E_MachineState.IMMEDIATE_STOPPED:	
	(* Move to System Initialising once there is no Immediate Fault *)
	IF GVL_MASTER.stMasterControl.bNoMachineImmediateFault  THEN	
		GVL_MASTER.stMachineStatus.eMachineState := E_MachineState.SYSTEM_INITIALISING;
	(* Move to Immediate Fault once there is an Immediate Fault *)
	ELSIF NOT GVL_MASTER.stMasterControl.bNoMachineImmediateFault THEN
		GVL_MASTER.stMachineStatus.eMachineState := E_MachineState.IMMEDIATE_FAULT;	
	END_IF
	
E_MachineState.SYSTEM_INITIALISING:		
	IF  GVL_MASTER.stMasterControl.bNoMachineImmediateFault	 AND GVL_MASTER.stMasterControl.bSystemInitialisingTimerComplete  THEN		
		GVL_MASTER.stMachineStatus.eMachineState := E_MachineState.SYSTEM_READY_TO_START;
	
	//Move to Cycle Stopped once there is a Cycle Stop Request AND All Stations are Cycle Stopped AND there is No Immediate Fault*)
	ELSIF GVL_HMI_GLOBAL.bStopButton
		OR (GVL_MASTER.stMasterControl.bNoMachineImmediateFault 
		AND (GVL_MASTER.stMasterControl.bSystemInitialisingTimeoutComplete OR GVL_MASTER.stMasterControl.bCycleStopRequest) AND GVL_MASTER.stMasterControl.bAllStationsCycledStopped)
	THEN		
		GVL_MASTER.stMachineStatus.eMachineState := E_MachineState.CYCLE_STOPPED;			
	ELSIF GVL_MASTER.stMasterControl.bNoMachineImmediateFault AND NOT GVL_MASTER.stMasterControl.bNoCycleStopFault THEN		
		GVL_MASTER.stMachineStatus.eMachineState := E_MachineState.CYCLE_STOP_FAULT;	
	ELSIF NOT GVL_MASTER.stMasterControl.bNoStationImmediateFault THEN
         GVL_MASTER.stMachineStatus.eMachineState := E_MachineState.IMMEDIATE_FAULT;
      	
	END_IF
	
E_MachineState.SYSTEM_READY_TO_START:
	bMemoSystemReadyToStart := TRUE;
	
	//Move to System Auto if the Start Button has been pressed
	IF GVL_MASTER.stMasterControl.bManualModeRequest THEN
		GVL_MASTER.stMachineStatus.eMachineState := E_MachineState.MANUAL_MODE;
	
	ELSIF GVL_HMI_GLOBAL.bStopButton THEN
        GVL_MASTER.stMachineStatus.eMachineState := E_MachineState.STOPPING; 
	ELSIF GVL_HMI_GLOBAL.bStartButton AND NOT PRG_Mastercycle.biClamp AND NOT PRG_Mastercycle.biPartPresent  THEN		//**LAA 18092025	
		GVL_MASTER.stMachineStatus.eMachineState := E_MachineState.SYSTEM_AUTO_CYCLE;
		
	//Move to Cycle Stopped once there is a Cycle Stop Request AND All Stations are Cycle Stopped AND there is No Immediate Fault
	ELSIF (GVL_MASTER.stMasterControl.bCycleStopRequest OR NOT	GVL_MASTER.stMasterControl.bNoCycleStopFault) 
	AND GVL_MASTER.stMasterControl.bNoMachineImmediateFault
	THEN				
		GVL_MASTER.stMachineStatus.eMachineState := E_MachineState.CYCLE_STOPPED;	
	ELSIF NOT GVL_MASTER.stMasterControl.bNoCycleStopFault THEN
		GVL_MASTER.stMachineStatus.eMachineState := E_MachineState.CYCLE_STOP_FAULT;
	ELSIF NOT GVL_MASTER.stMasterControl.bNoMachineImmediateFault OR NOT GVL_MASTER.stMasterControl.bNoStationImmediateFault THEN
       GVL_MASTER.stMachineStatus.eMachineState := E_MachineState.IMMEDIATE_FAULT ;	
	   
	END_IF
	

	
	
	
E_MachineState.SYSTEM_AUTO_CYCLE:	
	//Move to System Dwell once there is a Dwell Request
	IF GVL_MASTER.stMasterControl.bDwellRequest THEN
		GVL_MASTER.stMachineStatus.eMachineState := E_MachineState.SYSTEM_DWELL;
	
	//Move to Cycle Stopped once there is a Cycle Stop Request AND All Stations are Cycle Stopped AND there is No Immediate Fault OR when cycle done
	ELSIF NOT GVL_MASTER.stMasterControl.bNoCycleStopFault THEN //Fast cycle stop	
		GVL_MASTER.stMachineStatus.eMachineState := E_MachineState.CYCLE_STOP_FAULT;
	(*ELSIF GVL_Master.bMachineCycleDone   THEN 
	stMachineStatus.eMachineState := E_MachineState.CYCLE_STOPPED; //Instant cycle stop???		*)
	ELSIF GVL_HMI_GLOBAL.bStopButton OR GVL_MASTER.stMasterControl.bCycleStopRequest OR GVL_HMI_GLOBAL.nRegionMain <> 1 THEN
		GVL_MASTER.stMachineStatus.eMachineState := E_MachineState.STOPPING; //Stopping sequence 
	ELSIF NOT GVL_MASTER.stMasterControl.bNoStationImmediateFault OR NOT GVL_MASTER.stMasterControl.bNoMachineImmediateFault THEN
		GVL_MASTER.stMachineStatus.eMachineState := E_MachineState.IMMEDIATE_FAULT;
	END_IF	

E_MachineState.SYSTEM_DWELL:		
	(* Move to System Auto Cycle once the Start Button is Pressed AND there is No Dwell Request *)
	IF NOT GVL_MASTER.stMasterControl.bDwellRequest THEN
		GVL_MASTER.stMachineStatus.eMachineState := E_MachineState.SYSTEM_AUTO_CYCLE;	
	(* Move to Cycle Stopped once there is a Cycle Stop Request AND All Stations are Cycle Stopped AND there is No Immediate Fault*)
	ELSIF (GVL_MASTER.stMasterControl.bCycleStopRequest OR	NOT	GVL_MASTER.stMasterControl.bNoCycleStopFault) 
		AND GVL_MASTER.stMasterControl.bAllStationsCycledStopped AND GVL_MASTER.stMasterControl.bNoMachineImmediateFault
	THEN				
		GVL_MASTER.stMachineStatus.eMachineState := E_MachineState.CYCLE_STOPPED;	
	END_IF

E_MachineState.STOPPING: 
	IF  GVL_MASTER.stMasterControl.bAllStationsCycledStopped THEN
		GVL_MASTER.stMachineStatus.eMachineState := E_MachineState.CYCLE_STOPPED;
	ELSIF NOT GVL_MASTER.stMasterControl.bNoCycleStopFault THEN
		GVL_MASTER.stMachineStatus.eMachineState := E_MachineState.CYCLE_STOP_FAULT;
	ELSIF NOT GVL_MASTER.stMasterControl.bNoMachineImmediateFault OR NOT GVL_MASTER.stMasterControl.bNoStationImmediateFault THEN
        GVL_MASTER.stMachineStatus.eMachineState := E_MachineState.IMMEDIATE_FAULT ;
	END_IF
	
E_MachineState.CYCLE_STOPPED:
	IF GVL_MASTER.stMasterControl.bManualModeRequest THEN
		GVL_MASTER.stMachineStatus.eMachineState := E_MachineState.MANUAL_MODE;			
	(* Move to System Initialising once there is no Cycle Stop Fault AND the Reset Button is Pressed *)
	ELSIF (GVL_MASTER.stMasterControl.bNoCycleStopFault AND GVL_HMI_GLOBAL.bResetButton )THEN
		GVL_MASTER.stMachineStatus.eMachineState := E_MachineState.SYSTEM_INITIALISING;		
	ELSIF NOT GVL_MASTER.stMasterControl.bNoStationImmediateFault THEN
       	GVL_MASTER.stMachineStatus.eMachineState := E_MachineState.IMMEDIATE_FAULT;
	END_IF	

E_MachineState.CYCLE_STOP_FAULT:	
	(* Move to Cycle Stopped once there no Cycle Stop Fault AND there is No Immediate Fault*)
	IF GVL_MASTER.stMasterControl.bNoCycleStopFault THEN
		GVL_MASTER.stMachineStatus.eMachineState := E_MachineState.CYCLE_STOPPED;
	END_IF	
ELSE 	
	GVL_MASTER.stMachineStatus.eMachineState := E_MachineState.SYSTEM_POWER_UP;	
	
E_MachineState.MANUAL_MODE:

	IF NOT GVL_MASTER.stMasterControl.bManualModeRequest THEN
		GVL_MASTER.stMachineStatus.eMachineState := E_MachineState.CYCLE_STOPPED;
	END_IF
	
E_MachineState.IMMEDIATE_FAULT:		
	(* Move to Immediate Stopped once there is an Immediate Fault *)
	IF GVL_MASTER.stMasterControl.bNoMachineImmediateFault AND  GVL_MASTER.stMasterControl.bNoStationImmediateFault THEN
		GVL_MASTER.stMachineStatus.eMachineState := E_MachineState.IMMEDIATE_STOPPED;		

	END_IF
END_CASE
//////////////////////////////////////////////////////////////////////////////////////////////////////////////
								//CYCLE STOP REQUEST//
//////////////////////////////////////////////////////////////////////////////////////////////////////////////
IF GVL_MASTER.stAlarms[0].bCycleStopRequest OR GVL_MASTER.stAlarms[1].bCycleStopRequest OR GVL_MASTER.stAlarms[2].bCycleStopRequest THEN
				GVL_MASTER.stMasterControl.bCycleStopRequest	:=	TRUE;
ELSE			GVL_MASTER.stMasterControl.bCycleStopRequest	:=	FALSE;
END_IF




(************************************* write all system states to variables ***********************)

GVL_MASTER.stMachineStatus.bSystemPowerUp :=(GVL_MASTER.stMachineStatus.eMachineState = E_MachineState.SYSTEM_POWER_UP);
GVL_MASTER.stMachineStatus.bImmediateStopped :=(GVL_MASTER.stMachineStatus.eMachineState = E_MachineState.IMMEDIATE_STOPPED);
GVL_MASTER.stMachineStatus.bSystemInitialising :=(GVL_MASTER.stMachineStatus.eMachineState = E_MachineState.SYSTEM_INITIALISING);
GVL_MASTER.stMachineStatus.bSystemReadyToStart := (GVL_MASTER.stMachineStatus.eMachineState = E_MachineState.SYSTEM_READY_TO_START);
GVL_MASTER.stMachineStatus.bSystemAutoCycle := (GVL_MASTER.stMachineStatus.eMachineState = E_MachineState.SYSTEM_AUTO_CYCLE);
GVL_MASTER.stMachineStatus.bSystemDwell := (GVL_MASTER.stMachineStatus.eMachineState = E_MachineState.SYSTEM_DWELL);
GVL_MASTER.stMachineStatus.bSystemStopping := (GVL_MASTER.stMachineStatus.eMachineState = E_MachineState.STOPPING);
GVL_MASTER.stMachineStatus.bCycleStopped := (GVL_MASTER.stMachineStatus.eMachineState = E_MachineState.CYCLE_STOPPED);
GVL_MASTER.stMachineStatus.bManualMode := (GVL_MASTER.stMachineStatus.eMachineState = E_MachineState.MANUAL_MODE);
GVL_MASTER.stMachineStatus.bImmediateFault := (GVL_MASTER.stMachineStatus.eMachineState = E_MachineState.IMMEDIATE_FAULT);
GVL_MASTER.stMachineStatus.bCycleStopFault := (GVL_MASTER.stMachineStatus.eMachineState = E_MachineState.CYCLE_STOP_FAULT);

ACTION ACT_MachineStatusBaner:
//Machine status banner action
//SYSTEM POWER UP
IF GVL_MASTER.stMachineStatus.bSystemPowerUp THEN	
	GVL_MASTER.stMachineStatus.sMachineStatusText := 'SYSTEM POWER UP';		// fill colour WHITE, text colour BLACK
	GVL_MASTER.stMachineStatus.nMachineStatusColour := nWHITE;
	GVL_MASTER.stMachineStatus.nMachineStatusTxtCol := nBLACK;
	GVL_MASTER.stMachineStatus.sBannerBckColor := sWHITE;
	GVL_MASTER.stMachineStatus.sBannerTextColor := sBLACK;
END_IF

(* IMMEDIATE STOPPED *)
IF GVL_MASTER.stMachineStatus.bImmediateStopped THEN	
	GVL_MASTER.stMachineStatus.sMachineStatusText := 'IMMEDIATE STOPPED';		// fill colour BLACK, text colour WHITE
	GVL_MASTER.stMachineStatus.nMachineStatusColour := nBLACK;
	GVL_MASTER.stMachineStatus.nMachineStatusTxtCol := nWHITE;
	GVL_MASTER.stMachineStatus.sBannerBckColor := sBLACK;
	GVL_MASTER.stMachineStatus.sBannerTextColor := sWHITE;	
END_IF

(* SYSTEM INITIALISING *)
IF GVL_MASTER.stMachineStatus.bSystemInitialising THEN	
	GVL_MASTER.stMachineStatus.sMachineStatusText := 'SYSTEM INITIALIZING';		// fill colour YELLOW, text colour BLACK
	GVL_MASTER.stMachineStatus.nMachineStatusColour := nYELLOW;
	GVL_MASTER.stMachineStatus.nMachineStatusTxtCol := nBLACK;
	GVL_MASTER.stMachineStatus.sBannerBckColor := sYELLOW;
	GVL_MASTER.stMachineStatus.sBannerTextColor := sBLACK;
END_IF
(*
(* SYSTEM IN STANDBY *)
IF stMachineStatus.bSystemStandby THEN
	stMachineStatus.sMachineStatusText := 'SYSTEM IN STANDBY';
	stMachineStatus.nMachineStatusColour := nORANGE;
	stMachineStatus.nMachineStatusTxtCol := nWHITE;
END_IF
*)
(* SYSTEM READY TO START FLASH ON *)
IF GVL_MASTER.stMachineStatus.bSystemReadyToStart AND GVL_MASTER.bFlash1Hz THEN
	GVL_MASTER.stMachineStatus.sMachineStatusText := 'SYSTEM READY TO START';		// fill colour GREEN, text colour WHITE
	GVL_MASTER.stMachineStatus.nMachineStatusColour := nGREEN;
	GVL_MASTER.stMachineStatus.nMachineStatusTxtCol := nWHITE;
	GVL_MASTER.stMachineStatus.sBannerBckColor := sGREEN;
	GVL_MASTER.stMachineStatus.sBannerTextColor := sWHITE;
END_IF

(* SYSTEM READY TO START FLASH OFF *)
IF GVL_MASTER.stMachineStatus.bSystemReadyToStart AND NOT GVL_MASTER.bFlash1Hz THEN	
	GVL_MASTER.stMachineStatus.sMachineStatusText := 'SYSTEM READY TO START';		// fill colour WHITE, text colour GREEN
	GVL_MASTER.stMachineStatus.nMachineStatusColour := nWHITE;
	GVL_MASTER.stMachineStatus.nMachineStatusTxtCol := nGREEN;
	GVL_MASTER.stMachineStatus.sBannerBckColor := sWHITE;
	GVL_MASTER.stMachineStatus.sBannerTextColor := sGREEN;
END_IF

(* SYSTEM AUTO CYCLE *)
IF GVL_MASTER.stMachineStatus.bSystemAutoCycle THEN	
	GVL_MASTER.stMachineStatus.sMachineStatusText := 'SYSTEM AUTO CYCLE';		// fill colour GREEN, text colour WHITE
	GVL_MASTER.stMachineStatus.nMachineStatusColour := nGREEN;
	GVL_MASTER.stMachineStatus.nMachineStatusTxtCol := nWHITE;
	GVL_MASTER.stMachineStatus.sBannerBckColor := sGREEN;
	GVL_MASTER.stMachineStatus.sBannerTextColor := sWHITE;	
END_IF

(* SYSTEM DWELL *)
IF GVL_MASTER.stMachineStatus.bSystemDwell THEN	
	GVL_MASTER.stMachineStatus.sMachineStatusText := 'SYSTEM DWELL';		// fill colour ORANGE, text colourWHITE
	GVL_MASTER.stMachineStatus.nMachineStatusColour := nORANGE;
	GVL_MASTER.stMachineStatus.nMachineStatusTxtCol := nWHITE;
	GVL_MASTER.stMachineStatus.sBannerBckColor := sORANGE;
	GVL_MASTER.stMachineStatus.sBannerTextColor := sWHITE;	
END_IF

(* STOPPING *)
IF GVL_MASTER.stMachineStatus.bSystemStopping AND GVL_MASTER.bFlash1Hz THEN	
	GVL_MASTER.stMachineStatus.sMachineStatusText := 'STOPPING';		// fill colour BLACK, text colour WHITE
	GVL_MASTER.stMachineStatus.nMachineStatusColour := nBLACK;
	GVL_MASTER.stMachineStatus.nMachineStatusTxtCol := nWHITE;
	GVL_MASTER.stMachineStatus.sBannerBckColor := sBLACK;
	GVL_MASTER.stMachineStatus.sBannerTextColor := sWHITE;	
END_IF

(* STOPPING *)
IF GVL_MASTER.stMachineStatus.bSystemStopping AND NOT GVL_MASTER.bFlash1Hz THEN	
	GVL_MASTER.stMachineStatus.sMachineStatusText := 'STOPPING';		// fill colour WHITE, text colour BLACK
	GVL_MASTER.stMachineStatus.nMachineStatusColour := nWHITE;
	GVL_MASTER.stMachineStatus.nMachineStatusTxtCol := nBLACK;
	GVL_MASTER.stMachineStatus.sBannerBckColor := sWHITE;
	GVL_MASTER.stMachineStatus.sBannerTextColor := sBLACK;	
END_IF

(* CYCLE STOPPED *)
IF GVL_MASTER.stMachineStatus.bCycleStopped THEN	
	GVL_MASTER.stMachineStatus.sMachineStatusText := 'CYCLE STOPPED';		// fill colour BLACK, text colour WHITE
	GVL_MASTER.stMachineStatus.nMachineStatusColour := nBLACK;
	GVL_MASTER.stMachineStatus.nMachineStatusTxtCol := nWHITE;
	GVL_MASTER.stMachineStatus.sBannerBckColor := sBLACK;
	GVL_MASTER.stMachineStatus.sBannerTextColor := sWHITE;	
END_IF

(* IMMEDIATE FAULT FLASH ON *)
IF GVL_MASTER.stMachineStatus.bImmediateFault AND GVL_MASTER.bFlash1Hz THEN	
	GVL_MASTER.stMachineStatus.sMachineStatusText := 'IMMEDIATE FAULT';		// fill colour RED, text colour WHITE
	GVL_MASTER.stMachineStatus.nMachineStatusColour := nRED;
	GVL_MASTER.stMachineStatus.nMachineStatusTxtCol := nWHITE;
	GVL_MASTER.stMachineStatus.sBannerBckColor := sRED;
	GVL_MASTER.stMachineStatus.sBannerTextColor := sWHITE;	
END_IF

(* IMMEDIATE FAULT FLASH OFF *)
IF GVL_MASTER.stMachineStatus.bImmediateFault AND NOT GVL_MASTER.bFlash1Hz THEN	
	GVL_MASTER.stMachineStatus.sMachineStatusText := 'IMMEDIATE FAULT';		// fill colour WHITE, text colour BLACK
	GVL_MASTER.stMachineStatus.nMachineStatusColour := nWHITE;
	GVL_MASTER.stMachineStatus.nMachineStatusTxtCol := nBLACK;
	GVL_MASTER.stMachineStatus.sBannerBckColor := sWHITE;
	GVL_MASTER.stMachineStatus.sBannerTextColor := sBLACK;	
END_IF

(* CYCLE STOP FAULT FLASH ON *)
IF GVL_MASTER.stMachineStatus.bCycleStopFault AND GVL_MASTER.bFlash1Hz THEN	
	GVL_MASTER.stMachineStatus.sMachineStatusText := 'CYCLE STOP FAULT';		// fill colour RED, text colour WHITE
	GVL_MASTER.stMachineStatus.nMachineStatusColour := nRED;
	GVL_MASTER.stMachineStatus.nMachineStatusTxtCol := nWHITE;
	GVL_MASTER.stMachineStatus.sBannerBckColor := sRED;
	GVL_MASTER.stMachineStatus.sBannerTextColor := sWHITE;	
END_IF

(* CYCLE STOP FAULT FLASH OFF *)
IF GVL_MASTER.stMachineStatus.bCycleStopFault AND NOT GVL_MASTER.bFlash1Hz THEN	
	GVL_MASTER.stMachineStatus.sMachineStatusText := 'CYCLE STOP FAULT';		// fill colour WHITE, text colour RED
	GVL_MASTER.stMachineStatus.nMachineStatusColour := nWHITE;
	GVL_MASTER.stMachineStatus.nMachineStatusTxtCol := nRED;
	GVL_MASTER.stMachineStatus.sBannerBckColor := sWHITE;
	GVL_MASTER.stMachineStatus.sBannerTextColor := sRED;	
END_IF

(* MANUAL MODE *)
IF GVL_MASTER.stMachineStatus.bManualMode THEN	
	GVL_MASTER.stMachineStatus.sMachineStatusText := 'MANUAL MODE';		// fill colour BLUE text colour WHITE
	GVL_MASTER.stMachineStatus.nMachineStatusColour := nBLUE;
	GVL_MASTER.stMachineStatus.nMachineStatusTxtCol := nWHITE;
	GVL_MASTER.stMachineStatus.sBannerBckColor := sBLUE;
	GVL_MASTER.stMachineStatus.sBannerTextColor := sWHITE;	
END_IF

(*
(* SYSTEM READY TO START FLASH ON *)
IF stMachineStatus.bSystemPurge AND bFlash1Hz THEN
	stMachineStatus.sMachineStatusText := 'SYSTEM PURGE';		// fill colour GREEN, text colour WHITE
	stMachineStatus.nMachineStatusColour := nORANGE;
	stMachineStatus.nMachineStatusTxtCol := nBLACK;
	stMachineStatus.sBannerBckColor := sORANGE;
	stMachineStatus.sBannerTextColor := sBLACK;	
END_IF

(* SYSTEM READY TO START FLASH OFF *)
IF stMachineStatus.bSystemPurge AND NOT bFlash1Hz THEN	
	stMachineStatus.sMachineStatusText := 'SYSTEM PURGE';		// fill colour WHITE, text colour GREEN
	stMachineStatus.nMachineStatusColour := nWHITE;
	stMachineStatus.nMachineStatusTxtCol := nBLUE;
	stMachineStatus.sBannerBckColor := sWHITE;
	stMachineStatus.sBannerTextColor := sBLUE;	
END_IF
*)
(*
(* CALIBRATION *)
IF stMachineStatus.bCalibrationFlag AND bFlash1Hz THEN	
	stMachineStatus.sMachineStatusText := 'CALIBRATION MODE';		// fill colour BLUE text colour WHITE
	stMachineStatus.nMachineStatusColour := nBLUE;
	stMachineStatus.nMachineStatusTxtCol := nWHITE;
	stMachineStatus.sBannerBckColor := sBLUE;
	stMachineStatus.sBannerTextColor := sWHITE;	
END_IF
IF stMachineStatus.bCalibrationFlag AND NOT bFlash1Hz THEN	
	stMachineStatus.sMachineStatusText := 'CALIBRATION MODE';		// fill colour BLUE text colour WHITE
	stMachineStatus.nMachineStatusColour := nWHITE;
	stMachineStatus.nMachineStatusTxtCol := nBLUE;
	stMachineStatus.sBannerBckColor := sWHITE;
	stMachineStatus.sBannerTextColor := sBLUE;	
END_IF
*)
END_ACTION

ACTION ACT_ManualMode:
IF	 GVL_MASTER.stMachineStatus.bSystemReadyToStart THEN
	GVL_HMI_GLOBAL.bEnableManualMode := TRUE;
ELSE GVL_HMI_GLOBAL.bEnableManualMode := FALSE;
END_IF


rtrigManualMode(CLK:= GVL_HMI_GLOBAL.nRegionMain=10);
rtrigManualModeOFF[1](CLK:=GVL_Master.stMachineStatus.bManualMode AND (GVL_HMI_GLOBAL.nRegionMain <> 10));
rtrigManualModeOFF[2](CLK:=GVL_Master.stMachineStatus.bManualMode AND GVL_HMI_GLOBAL.bStopButton);
rtrigManualModeOFF[3](CLK:=GVL_Master.stMachineStatus.bManualMode AND NOT GVL_Master.stMasterControl.bNoStationImmediateFault );
rtrigManualModeOff[4](CLK := GVL_HMI_GLOBAL.bManualModeOff[1], Q => GVL_HMI_GLOBAL.bManualModeOff[2]);

IF rtrigManualMode.Q THEN 
	GVL_Master.stMasterControl.bManualModeRequest := TRUE;
	GVL_HMI_GLOBAL.bManualModeOff[1] := FALSE;
ELSIF rtrigManualModeOFF[1].Q OR rtrigManualModeOFF[2].Q OR rtrigManualModeOFF[3].Q THEN
	GVL_Master.stMasterControl.bManualModeRequest := FALSE ;
	GVL_HMI_GLOBAL.bManualModeOff[1] := TRUE;
	
ELSE GVL_HMI_GLOBAL.bManualModeOff[1] := FALSE;
	
END_IF





IF GVL_Master.stMachineStatus.bManualMode  THEN
	GVL_Master.stStationSruct[1].bStationManualRequestHMI := TRUE;
	GVL_Master.stStationSruct[2].bStationManualRequestHMI := TRUE;
ELSE
    GVL_Master.stStationSruct[1].bStationManualRequestHMI := FALSE;
	GVL_Master.stStationSruct[2].bStationManualRequestHMI := FALSE;
END_IF
END_ACTION

ACTION ACT_MasterTime:
//Aux functions call
tonTimeUpdateGen(	IN := NOT bUpdateSysTime,
					PT := tSysTimeUpdatePeriod,
					Q => bUpdateSysTime);

//bReadyToRead :=  Tc2_System.MEMCMP( ADR( stTimeStamp), ADR (stNullTimeStamp), SIZEOF(stTimeStamp)) <> 0 AND NOT  fbGetSystemTime.BUSY;	
			(*keczi*)	(*zrobione po to zeby w wypadku jak po starcie PLC na HMI mial pokazywac czas alarmu '00:00:00', zebyb poczekal az faktycznie pokazuje date i czas*)

//Get Current System Time
fbGetSystemTime(NETID := ,
				START := bFirstScan OR bUpdateSysTime,
				TMOUT := ,
				BUSY => ,
				ERR => ,
				ERRID => ,
				TIMESTR => );
				
//Get system time done detection - one-shot
rtrigSysTimeCollected(CLK := NOT fbGetSystemTime.BUSY);

//Synchronize Real-Time clock with system time
fbRTClock(	EN := rtrigSysTimeCollected.Q, 
			PDT := fbGetSystemTime.TIMESTR,
			CDT => stTimeStamp, 
			Q => bReadyToRead);

// System Date and Time in Proper Order 
IF bReadyToRead THEN
	sRawDateTime := SYSTEMTIME_TO_STRING(stTimeStamp);  // format: YYYY-MM-DD-hh:mm:ss.xxx
	GVL_HMI_GLOBAL.sSystemDate := CONCAT(CONCAT(CONCAT(CONCAT(MID(sRawDateTime, 2, 9), '.'),  MID(sRawDateTime, 2, 6)), '.'), LEFT(sRawDateTime, 4));
	GVL_HMI_GLOBAL.sSystemTime := MID(sRawDateTime, 8, 12);
	sDateTime := CONCAT(CONCAT(GVL_HMI_GLOBAL.sSystemDate, '  '), GVL_HMI_GLOBAL.sSystemTime);
	sDateTimeSpaces	:= CONCAT(sDateTime, '    ');
END_IF;

bFirstScan := FALSE;
END_ACTION

END_PROGRAM

// ---- POUs/E_HMI/PRG_HMI.TcPOU
PROGRAM PRG_HMI
VAR
	

	tonCaseDelay				: ARRAY [1..20] OF TON;
	tofCase						: ARRAY [1..20] OF TOF;
	rtrigCaseTriger				: ARRAY [1..20] OF R_TRIG;
	rsCase						: ARRAY [1..10] OF RS;
	
	fbWritePersistentData		:FB_WritePersistentData;
	fWritePersistentData		: F_TRIG;
	
	tonResetStatistics			: TON;
	

END_VAR

ACT_ScreensNamesSet();
ACT_Buttons();
ACT_TimTrig();
ACT_General();
ACT_SavePersistentVariables();

tonResetStatistics( IN := 	GVL_HMI_GLOBAL.aResetHeightSensorBadParts [1] 	OR
							GVL_HMI_GLOBAL.aResetHeightSensorBadParts [2] 	OR
							GVL_HMI_GLOBAL.aResetHeightSensorBadParts [3] 	OR
							GVL_HMI_GLOBAL.aResetHeightSensorBadParts [4] 	OR
							GVL_HMI_GLOBAL.aResetHeightSensorGoodParts[1]	OR
							GVL_HMI_GLOBAL.aResetHeightSensorGoodParts[2]	OR
							GVL_HMI_GLOBAL.aResetHeightSensorGoodParts[3]	OR
							GVL_HMI_GLOBAL.aResetHeightSensorGoodParts[4]	OR
							GVL_HMI_GLOBAL.bResetHeightFailParts			OR
							GVL_HMI_GLOBAL.bResetHeightGoodParts			OR
							GVL_HMI_GLOBAL.bResetGoodParts					OR
							GVL_HMI_GLOBAL.bResetLeakBadParts				OR
							GVL_HMI_GLOBAL.bResetLeakGoodParts				OR
							GVL_HMI_GLOBAL.bResetFailedParts				OR
							GVL_HMI_GLOBAL.bResetGoodParts					,
							PT												:= T#500MS);

ACTION ACT_Buttons:
ACT_TimTrig();

IF tonCaseDelay[1].Q THEN
	
		GVL_HMI_GLOBAL.bResetButton	:= FALSE;
		
END_IF
IF tonCaseDelay[2].Q THEN
	
		GVL_HMI_GLOBAL.bStopButton	:= FALSE;
		
END_IF
IF tonCaseDelay[3].Q THEN
	
		GVL_HMI_GLOBAL.bStartButton	:= FALSE;
		
END_IF

IF GVL_HMI_GLOBAL.bStartLeakMan THEN
	GVL_IO.dw_B07_i28General_I_O.bStart := TRUE;
END_IF
IF tonCaseDelay[4].Q THEN
	
		GVL_HMI_GLOBAL.bStartLeakMan	:= FALSE;
		GVL_IO.dw_B07_i28General_I_O.bStart := FALSE;
END_IF

IF GVL_HMI_GLOBAL.bStopLeakMan THEN
	GVL_IO.dw_B07_i28General_I_O.bStop := TRUE;
END_IF
IF tonCaseDelay[5].Q THEN
	
		GVL_HMI_GLOBAL.bStopLeakMan	:= FALSE;
		GVL_IO.dw_B07_i28General_I_O.bStop := FALSE;
		
END_IF

IF GVL_HMI_GLOBAL.bResetLeakMan THEN
	GVL_IO.dw_B07_i28General_I_O.bReset := TRUE;
END_IF
IF tonCaseDelay[6].Q THEN
	
		GVL_HMI_GLOBAL.bResetLeakMan	:= FALSE;
		GVL_IO.dw_B07_i28General_I_O.bReset := FALSE;
		
END_IF

IF tonCaseDelay[7].Q THEN
	
		GVL_HMI_GLOBAL.bShutDown	:= FALSE;
		
END_IF
IF tonCaseDelay[8].Q THEN
	
		GVL_HMI_GLOBAL.bSetLeakProgramID	:= FALSE;
		
END_IF

IF tonCaseDelay[9].Q THEN
	
		GVL_HMI_GLOBAL.bSetSetPointsHeightTest	:= FALSE;
		
END_IF


							
IF tonResetStatistics.Q THEN
	
							GVL_HMI_GLOBAL.aResetHeightSensorBadParts [1] 	:= FALSE;
							GVL_HMI_GLOBAL.aResetHeightSensorBadParts [2] 	:= FALSE;
							GVL_HMI_GLOBAL.aResetHeightSensorBadParts [3] 	:= FALSE;
							GVL_HMI_GLOBAL.aResetHeightSensorBadParts [4] 	:= FALSE;
							GVL_HMI_GLOBAL.aResetHeightSensorGoodParts[1]	:= FALSE;
							GVL_HMI_GLOBAL.aResetHeightSensorGoodParts[2]	:= FALSE;
							GVL_HMI_GLOBAL.aResetHeightSensorGoodParts[3]	:= FALSE;
							GVL_HMI_GLOBAL.aResetHeightSensorGoodParts[4]	:= FALSE;
							GVL_HMI_GLOBAL.bResetHeightFailParts			:= FALSE;
							GVL_HMI_GLOBAL.bResetHeightGoodParts			:= FALSE;
							GVL_HMI_GLOBAL.bResetGoodParts					:= FALSE;
							GVL_HMI_GLOBAL.bResetLeakBadParts				:= FALSE;
							GVL_HMI_GLOBAL.bResetLeakGoodParts				:= FALSE;
							GVL_HMI_GLOBAL.bResetFailedParts				:= FALSE;
							GVL_HMI_GLOBAL.bResetGoodParts					:= FALSE;


END_IF
END_ACTION

ACTION ACT_General:

IF tofCase[1].Q AND 
( NOT GVL_MASTER.stMasterControl.bNoStationImmediateFault OR NOT GVL_MASTER.stMasterControl.bNoCycleStopFault) THEN
	GVL_HMI_GLOBAL.bAutocycleFaultDialog := TRUE;
END_IF
END_ACTION

ACTION ACT_SavePersistentVariables:
fWritePersistentData(CLK := GVL_HMI_GLOBAL.nRegionMain = 5);

fbWritePersistentData(	PORT 				:= 851,
						START 				:= fWritePersistentData.Q,);
END_ACTION

ACTION ACT_ScreensNamesSet:
GVL_HMI_GLOBAL.aIOScreen[0] := 'Overview';
GVL_HMI_GLOBAL.aIOScreen[1] := 'HMI - CP2913-0000 | Beckhoff HMI';
GVL_HMI_GLOBAL.aIOScreen[2] := 'PLC - C6015-0010 | Beckhoff PLC | Windows 10 Embedded';
GVL_HMI_GLOBAL.aIOScreen[3] := 'Terminal 1- EK1100 | EtherCAT Coupler';
GVL_HMI_GLOBAL.aIOScreen[4] := 'Terminal 2 - EL6070 | Licence ';
GVL_HMI_GLOBAL.aIOScreen[5] := CONCAT('Terminal 3 - ' , GVL_IO.dw_T02_EL1809.sTerminalName);
GVL_HMI_GLOBAL.aIOScreen[6] := CONCAT('Terminal 4 - ' , GVL_IO.dw_T03_EL2809.sTerminalName);
GVL_HMI_GLOBAL.aIOScreen[7] := 'Terminal 12 - EL6631 |  2-port communication interface';
GVL_HMI_GLOBAL.aIOScreen[8] := 'DL-PN1 | Keyence Communication Unit | ProfiNET';
GVL_HMI_GLOBAL.aIOScreen[9] := 'I28 | Cincinnati Leak Tester | ProfiNET';


GVL_HMI_GLOBAL.aManualScreen[0] := 'Keyence | Height Test';
GVL_HMI_GLOBAL.aManualScreen[1] := 'Cincinnati | Leak Test';
END_ACTION

ACTION ACT_TimTrig:


tonCaseDelay[1](IN:= GVL_HMI_GLOBAL.bResetButton,PT:=T#500MS);
tonCaseDelay[2](IN:= GVL_HMI_GLOBAL.bStopButton,PT:=T#500MS);
tonCaseDelay[3](IN:= GVL_HMI_GLOBAL.bStartButton,PT:=T#500MS);
tonCaseDelay[4](IN:= GVL_HMI_GLOBAL.bStartLeakMan,PT:=T#500MS);
tonCaseDelay[5](IN:= GVL_HMI_GLOBAL.bStopLeakMan,PT:=T#500MS);
tonCaseDelay[6](IN:= GVL_HMI_GLOBAL.bResetLeakMan,PT:=T#500MS);
//tonCaseDelay[7](IN:= GVL_HMI_GLOBAL.bShutDown,PT:=T#500MS);
tonCaseDelay[8](IN:= GVL_HMI_GLOBAL.bSetLeakProgramID,PT:=T#5S);
tonCaseDelay[9](IN:= GVL_HMI_GLOBAL.bSetSetPointsHeightTest,PT:=T#1S);
tonCaseDelay[10](IN:= GVL_HMI_GLOBAL.bManualMeasureHeightTest,PT:=T#1S);
tonCaseDelay[11](IN:= ,PT:=T#500MS);
tonCaseDelay[12](IN:=,PT:=T#500MS);

tofCase[1](IN:= (GVL_Master.stStationSruct[0].nState > 1000 AND GVL_Master.stStationSruct[0].nState < 1900),PT:=T#1S);


rtrigCaseTriger[1](CLK := GVL_MASTER.stNest.bPieceReject);
END_ACTION

END_PROGRAM

// ---- POUs/C_LeakTest/PRG_LeakTestEvents_Info.TcPOU
PROGRAM PRG_LeakTestEvents_Info
VAR
	
	asLeakTesterSegments 				: ARRAY [0..200] OF WSTRING;
	asLeakTesterTestData 				: ARRAY [0..200] OF WSTRING;
	asLeakTesterUnit 	 				: ARRAY [0..200] OF WSTRING;
	asLeakTesterPrecision				: ARRAY [0..10]  OF WSTRING;
	asLeakTesterProgramEvaluation		: ARRAY [0..20]  OF WSTRING;
	asLeakTesterTestEvaluation			: ARRAY [0..150]  OF WSTRING;
	asLeakTesterTestType				: ARRAY [0..25]  OF WSTRING;
	fLeakTesterActive					: F_TRIG;
	bLeakTesterActive					: BOOL;
	Test1								: BOOL;
	
	i									: DINT;
	

END_VAR

ACT_LiveSegmentCode();
ACT_LeakTesterTestData();
ACT_LeakTesterUnit();
ACT_Precision();
ACT_ProgramEvaluation();
ACT_LeakTesterTestEvaluation();
ACT_TestType();

//Last Result DATA

GVL_IO.dw_B07_i28LastResult.sPartEvaluation 		:= asLeakTesterTestData[GVL_IO.dw_B07_i28LastResult.inTestType];
GVL_IO.dw_B07_i28LastResult.sPrecision				:= asLeakTesterPrecision[GVL_IO.dw_B07_i28LastResult.inPrecisionCode];
GVL_IO.dw_B07_i28LastResult.sTestType				:= asLeakTesterTestType[ GVL_IO.dw_B07_i28LastResult.inPartEvaluation];
GVL_IO.dw_B07_i28LastResult.sUnit1      			:= asLeakTesterUnit[GVL_IO.dw_B07_i28LastResult.inUnitCode1];
GVL_IO.dw_B07_i28LastResult.sUnit2					:= asLeakTesterUnit[GVL_IO.dw_B07_i28LastResult.inUnitCode2];
GVL_IO.dw_B07_i28LastResult.sVariable1				:= asLeakTesterTestData[GVL_IO.dw_B07_i28LastResult.inVariableCode1];
GVL_IO.dw_B07_i28LastResult.sVariable2				:= asLeakTesterTestData[GVL_IO.dw_B07_i28LastResult.inVariableCode2];

//Live DATA


GVL_IO.dw_B07_i28LiveMeasurement.sPrecision1		:= asLeakTesterPrecision[GVL_IO.dw_B07_i28LiveMeasurement.inPrecisionCode1];
GVL_IO.dw_B07_i28LiveMeasurement.sPrecision2		:= asLeakTesterPrecision[GVL_IO.dw_B07_i28LiveMeasurement.inPrecisionCode2];
GVL_IO.dw_B07_i28LiveMeasurement.sPrecision3		:= asLeakTesterPrecision[GVL_IO.dw_B07_i28LiveMeasurement.inPrecisionCode3];
GVL_IO.dw_B07_i28LiveMeasurement.sPrecision4		:= asLeakTesterPrecision[GVL_IO.dw_B07_i28LiveMeasurement.inPrecisionCode4];
GVL_IO.dw_B07_i28LiveMeasurement.sSegmentCode		:= asLeakTesterSegments[GVL_IO.dw_B07_i28LiveMeasurement.inSegmentCode];
GVL_IO.dw_B07_i28LiveMeasurement.sUnit1				:= asLeakTesterUnit[GVL_IO.dw_B07_i28LiveMeasureMENT.inUnitCode1];
GVL_IO.dw_B07_i28LiveMeasurement.sUnit2				:= asLeakTesterUnit[GVL_IO.dw_B07_i28LiveMeasureMENT.inUnitCode2];
GVL_IO.dw_B07_i28LiveMeasurement.sUnit3				:= asLeakTesterUnit[GVL_IO.dw_B07_i28LiveMeasureMENT.inUnitCode3];
GVL_IO.dw_B07_i28LiveMeasurement.sUnit4				:= asLeakTesterUnit[GVL_IO.dw_B07_i28LiveMeasureMENT.inUnitCode4];
GVL_IO.dw_B07_i28LiveMeasurement.sVariable1			:= asLeakTesterTestData[GVL_IO.dw_B07_i28LiveMeasurement.inVariableCode1];
GVL_IO.dw_B07_i28LiveMeasurement.sVariable2			:= asLeakTesterTestData[GVL_IO.dw_B07_i28LiveMeasurement.inVariableCode2];
GVL_IO.dw_B07_i28LiveMeasurement.sVariable3			:= asLeakTesterTestData[GVL_IO.dw_B07_i28LiveMeasurement.inVariableCode3];
GVL_IO.dw_B07_i28LiveMeasurement.sVariable4			:= asLeakTesterTestData[GVL_IO.dw_B07_i28LiveMeasurement.inVariableCode4];


ACT_LastResultSet();

ACTION ACT_LastResultSet:

fLeakTesterActive(CLK := GVL_IO.dw_B07_i28General_I_O.bTestActiveLiveData, Q => bLeakTesterActive);

IF bLeakTesterActive THEN
	
	FOR i :=200 TO 1 BY (-1) DO
		GVL_PERSIST.ast_i28LasResult[i]	:= GVL_PERSIST.ast_i28LasResult[i-1];
	END_FOR
	
	GVL_PERSIST.ast_i28LasResult[0] := GVL_IO.dw_B07_i28LastResult;
	GVL_PERSIST.ast_i28LasResult[0].sTime := GVL_HMI_GLOBAL.sSystemTime;
	GVL_PERSIST.ast_i28LasResult[0].sDate := GVL_HMI_GLOBAL.sSystemDate;

END_IF
END_ACTION

ACTION ACT_LeakTesterTestData:
asLeakTesterTestData[0] := "NO DATA";
asLeakTesterTestData[1] := "Elapsed Timer";
asLeakTesterTestData[2] := "Segment Timer";
asLeakTesterTestData[3] := "Test Execution Time";
asLeakTesterTestData[4] := "Target Pressure";
asLeakTesterTestData[5] := "Test Pressure";
asLeakTesterTestData[6] := "Master Part Profile Test Pressure";
asLeakTesterTestData[7] := "Master Part & Leak Profile Test Pressure";
asLeakTesterTestData[8] := "Leak Standard Calibrated Pressure";
asLeakTesterTestData[9] := "Self Test Pressure";
asLeakTesterTestData[10] := "Measured Pressure";
asLeakTesterTestData[11] := "Instrument Pressure";
asLeakTesterTestData[12] := "Master Gauge Pressure";
asLeakTesterTestData[13] := "Master Part Pressure Loss (Corrected)";
asLeakTesterTestData[14] := "Low Limit Pressure Loss";
asLeakTesterTestData[15] := "High Limit Pressure Loss";
asLeakTesterTestData[16] := "Master Part & Leak Pressure Loss (Corrected)";
asLeakTesterTestData[17] := "Pressure Loss (Corrected)";
asLeakTesterTestData[18] := "Pressure Loss (Actual Read)";
asLeakTesterTestData[19] := "Master Part Flow Offset (Corrected)";
asLeakTesterTestData[20] := "Performance Factor";
asLeakTesterTestData[21] := "Low Limit Rate";
asLeakTesterTestData[22] := "High Limit Rate";
asLeakTesterTestData[23] := "Loss Rate (Corrected)";
asLeakTesterTestData[24] := "Loss Rate (Actual Read)";
asLeakTesterTestData[25] := "Quik Test Pressure";
asLeakTesterTestData[26] := "Quik Test Loss (Corrected)";
asLeakTesterTestData[27] := "Quik Test Flow (Corrected)";
asLeakTesterTestData[28] := "Low Limit Leak Rate";
asLeakTesterTestData[29] := "High Limit Leak Rate";
asLeakTesterTestData[30] := "Predicted Leak Rate";
asLeakTesterTestData[31] := "Leak Rate";
asLeakTesterTestData[32] := "Corrected Leak Standard Calibrated Flow";
asLeakTesterTestData[33] := "Measured Flow";
asLeakTesterTestData[34] := "Environmental Drift Correction Offset";
asLeakTesterTestData[35] := "Transducer Type";
asLeakTesterTestData[36] := "Transducer Typical Residual";
asLeakTesterTestData[37] := "Transducer Zero Low Window";
asLeakTesterTestData[38] := "Transducer Zero High Window";
asLeakTesterTestData[39] := "Regulator Type";
asLeakTesterTestData[40] := "Analog A/D Value";
asLeakTesterTestData[41] := "Peak Pressure";
asLeakTesterTestData[42] := "Analog Input";
asLeakTesterTestData[43] := "Analog Output";
asLeakTesterTestData[44] := "Event Delta Pressure";
asLeakTesterTestData[45] := "Alternate Leak Rate";
asLeakTesterTestData[46] := "DP Master Part Pressure Loss (Corrected)";
asLeakTesterTestData[47] := "DP Master Part & Leak Pressure Loss (Corrected)";
asLeakTesterTestData[48] := "Master Part Quik Pressure Loss (Corrected)";
asLeakTesterTestData[49] := "Master Part Quik Pressure Loss (Actual Read)";
asLeakTesterTestData[50] := "Master Part & Leak Quik Pressure Loss (Corrected)";
asLeakTesterTestData[51] := "Master Part & Leak Quik Pressure Loss (Actual Read)";
asLeakTesterTestData[52] := "Master Part Quik Test Pressure";
asLeakTesterTestData[53] := "Master Part & Leak Quik Test Pressure";
asLeakTesterTestData[54] := "Master Part Quik DP Pressure Loss (Corrected)";
asLeakTesterTestData[55] := "Master Part Quik DP Pressure Loss (Actual Read)";
asLeakTesterTestData[56] := "Master Part & Leak Quik DP Pressure Loss (Actual Read)";
asLeakTesterTestData[57] := "Signal to Noise Ratio";
asLeakTesterTestData[58] := "Effective Number of Bits";
asLeakTesterTestData[59] := "Flicker Free Number of Bits";
asLeakTesterTestData[60] := "High Limit Percent Volume";
asLeakTesterTestData[61] := "Part Percent Volume";
asLeakTesterTestData[62] := "Reference Pressure";
asLeakTesterTestData[63] := "Fill Pressure";
asLeakTesterTestData[64] := "Transducer Cal/Verify - Number of Points";
asLeakTesterTestData[65] := "Transducer - Setpoint Pressure Value";
asLeakTesterTestData[66] := "Transducer - Instrument Pressure Reading";
asLeakTesterTestData[67] := "Transducer - Instrument Flow Reading";
asLeakTesterTestData[68] := "Transducer - Analog Value";
asLeakTesterTestData[69] := "Transducer - Master Reading";
asLeakTesterTestData[70] := "Transducer - Master Value";
asLeakTesterTestData[71] := "Transducer - Atmospheric Pressure";
asLeakTesterTestData[72] := "Transducer - Linearity";
asLeakTesterTestData[73] := "Electronic Regulator Cal - Number of Points";
asLeakTesterTestData[74] := "Electronic Regulator - Instrument Pressure Reading";
asLeakTesterTestData[75] := "Electronic Regulator - Analog Value";
asLeakTesterTestData[76] := "Electronic Regulator - Master Value";
asLeakTesterTestData[77] := "Electronic Regulator Analysis - Number of Points";
asLeakTesterTestData[78] := "Electronic Regulator Analysis - Instrument Pressure Reading";
asLeakTesterTestData[79] := "Electronic Regulator Analysis - Voltage Low Limit";
asLeakTesterTestData[80] := "Electronic Regulator Analysis - Voltage High Limit";
asLeakTesterTestData[81] := "Event Pressure";
asLeakTesterTestData[82] := "Part Flow";
asLeakTesterTestData[83] := "Pre-Pressure";
asLeakTesterTestData[84] := "Tracer Cumulative Leak Rate";
asLeakTesterTestData[85] := "Sniffer Test Location";
asLeakTesterTestData[86] := "Electronic Regulator Cal - Atmospheric Pressure";
asLeakTesterTestData[87] := "REF External Xdcr Pressure";
asLeakTesterTestData[88] := "Differential Pressure Loss (Corrected)";
asLeakTesterTestData[89] := "Differential Pressure Loss (Actual Read)";
asLeakTesterTestData[90] := "Reference Pressure Loss";
asLeakTesterTestData[91] := "Differential Pressure Loss (Actual Read)";
asLeakTesterTestData[92] := "Input State";
asLeakTesterTestData[93] := "Leak Loss";
asLeakTesterTestData[94] := "Batch Quantity";
asLeakTesterTestData[95] := "DP Leak Loss";
asLeakTesterTestData[96] := "Average Quantity";
asLeakTesterTestData[97] := "Charge Pressure";
asLeakTesterTestData[98] := "Standard Pressure";
asLeakTesterTestData[99] := "Instrument Volume";
asLeakTesterTestData[100] := "Part Volume";
asLeakTesterTestData[101] := "Test Measurement Time";
asLeakTesterTestData[102] := "Calculated Leak Rate Offset";
END_ACTION

ACTION ACT_LeakTesterTestEvaluation:
asLeakTesterTestEvaluation[0] := "NO DATA";
asLeakTesterTestEvaluation[1] := "PROGRAM ACCEPT";
asLeakTesterTestEvaluation[2] := "PROGRAM REJECT";
asLeakTesterTestEvaluation[3] := "PART REJECT - LEVEL 1";
asLeakTesterTestEvaluation[4] := "PART REJECT - LEVEL 2";
asLeakTesterTestEvaluation[5] := "PART REJECT - LEVEL 3";
asLeakTesterTestEvaluation[6] := "PROGRAM CALIBRATION PASSED";
asLeakTesterTestEvaluation[7] := "PROGRAM CALIBRATION FAILED";
asLeakTesterTestEvaluation[8] := "MASTER PART COMPLETE";
asLeakTesterTestEvaluation[9] := "SELF-TEST PASSED";
asLeakTesterTestEvaluation[10] := "SELF-TEST FAILED";
asLeakTesterTestEvaluation[11] := "SEQUENCE COMPLETE";
asLeakTesterTestEvaluation[12] := "SEVERE LEAK";
asLeakTesterTestEvaluation[13] := "TEST PRESSURE LOW";
asLeakTesterTestEvaluation[14] := "TEST PRESSURE HIGH";
asLeakTesterTestEvaluation[15] := "BELOW TARGET PRESSURE";
asLeakTesterTestEvaluation[16] := "ABOVE TARGET PRESSURE";
asLeakTesterTestEvaluation[17] := "HELIUM BACKGROUND FAULT";
asLeakTesterTestEvaluation[18] := "PART EVAC FAULT";
asLeakTesterTestEvaluation[19] := "TRANSDUCER ZERO BAD";
asLeakTesterTestEvaluation[20] := "TRANSDUCER OVER-RANGE";
asLeakTesterTestEvaluation[21] := "FLOW TRANSDUCER ZERO BAD";
asLeakTesterTestEvaluation[22] := "FLOW TRANSDUCER OVER-RANGE";
asLeakTesterTestEvaluation[23] := "ERROR: EXCESSIVE FLOW";
asLeakTesterTestEvaluation[24] := "PROGRAM CONFIGURATION ERROR";
asLeakTesterTestEvaluation[25] := "PROG ERROR";
asLeakTesterTestEvaluation[26] := "CALCULATION ERROR";
asLeakTesterTestEvaluation[27] := "INVALID PROGRAM SELECTED";
asLeakTesterTestEvaluation[28] := "INVALID CALIBRATION DATA";
asLeakTesterTestEvaluation[29] := "INVALID I/O CONFIGURATION";
asLeakTesterTestEvaluation[30] := "I/O FAULT";
asLeakTesterTestEvaluation[31] := "CAL REQUIRED - LIMIT EXCEEDED";
asLeakTesterTestEvaluation[32] := "CAL REQUIRED - PARAM CHANGED";
asLeakTesterTestEvaluation[33] := "MIN PERF FACTOR ERROR";
asLeakTesterTestEvaluation[34] := "MASTER+LEAK LOSS<MASTER LOSS";
asLeakTesterTestEvaluation[35] := "MASTER LOSS>MAX M+L LOSS";
asLeakTesterTestEvaluation[36] := "MASTER+LEAK LOSS>MAX M+L LOSS";
asLeakTesterTestEvaluation[37] := "MASTER FLOW>MAX M+L FLOW";
asLeakTesterTestEvaluation[38] := "MASTER FLOW<MIN MASTER FLOW";
asLeakTesterTestEvaluation[39] := "MASTER+LEAK FLOW>MAX M+L FLOW";
asLeakTesterTestEvaluation[40] := "MASTER FLOW>MAX MASTER FLOW";
asLeakTesterTestEvaluation[41] := "MASTER+LEAK FLOW>MAX MASTER FLOW";
asLeakTesterTestEvaluation[42] := "MASTER LOSS<MIN MASTER LOSS";
asLeakTesterTestEvaluation[43] := "MASTER LOSS>MAX MASTER LOSS";
asLeakTesterTestEvaluation[44] := "STOP BUTTON PRESSED";
asLeakTesterTestEvaluation[45] := "STOP INPUT RECEIVED";
asLeakTesterTestEvaluation[46] := "ERROR: STOP INPUT HIGH";
asLeakTesterTestEvaluation[47] := "START COMMON INPUT LOW";
asLeakTesterTestEvaluation[48] := "ERROR: ANTI-TIE DOWN";
asLeakTesterTestEvaluation[49] := "ERROR: PART NOT PRESENT";
asLeakTesterTestEvaluation[50] := "ERROR: PART NOT CHANGED";
asLeakTesterTestEvaluation[51] := "EXT SWITCH DID NOT GO LOW";
asLeakTesterTestEvaluation[52] := "EXT SWITCH DID NOT GO HIGH";
asLeakTesterTestEvaluation[53] := "ERROR: TOOLING NOT RESET";
asLeakTesterTestEvaluation[54] := "ERROR: TOOLING NOT EXTENDED";
asLeakTesterTestEvaluation[55] := "ERROR: TOOLING NOT RETRACTED";
asLeakTesterTestEvaluation[56] := "TOOLING RESET";
asLeakTesterTestEvaluation[57] := "ERROR: PART MARK FAULT";
asLeakTesterTestEvaluation[58] := "PART NOT FULL";
asLeakTesterTestEvaluation[59] := "PART NOT EXHAUSTED";
asLeakTesterTestEvaluation[60] := "PART NOT STABILIZED";
asLeakTesterTestEvaluation[61] := "AUTOSETUP SEQ COMPLETE";
asLeakTesterTestEvaluation[62] := "DP TRANSDUCER ZERO BAD";
asLeakTesterTestEvaluation[63] := "DP TRANSDUCER OVER-RANGE";
asLeakTesterTestEvaluation[64] := "ERROR: TWO-INPUT REQ TO START";
asLeakTesterTestEvaluation[65] := "ERROR: BARCODE REQ TO START";
asLeakTesterTestEvaluation[66] := "DP TRANSDUCER FAULT";
asLeakTesterTestEvaluation[67] := "ERROR: NO LINKS DEFINED";
asLeakTesterTestEvaluation[68] := "ERROR: LINK EXECUTION LOOP";
asLeakTesterTestEvaluation[69] := "ERROR: LINK PROG IS PARENT";
asLeakTesterTestEvaluation[70] := "ERROR: LINK PROG UNDEFINED";
asLeakTesterTestEvaluation[71] := "ERROR: DISSIMILAR LINK ORDER";
asLeakTesterTestEvaluation[72] := "ERROR: DUPLICATE TARGET LINK";
asLeakTesterTestEvaluation[73] := "CAL PROGRAM ACCEPT";
asLeakTesterTestEvaluation[74] := "CAL PROGRAM REJECT";
asLeakTesterTestEvaluation[75] := "PRESSURE TRANSDUCER FAULT";
asLeakTesterTestEvaluation[76] := "NO EVENT OCCURRED";
asLeakTesterTestEvaluation[77] := "SYSTEM PRESSURE EXCEEDED";
asLeakTesterTestEvaluation[78] := "PRESSURE SELECT CONFIG ERROR";
asLeakTesterTestEvaluation[79] := "LEAK STD SELECT CONFIG ERROR";
asLeakTesterTestEvaluation[80] := "VENT PART RESET TOOLING";
asLeakTesterTestEvaluation[81] := "TRANSDUCER CAL COMPLETE";
asLeakTesterTestEvaluation[82] := "TRANSDUCER CAL ERROR";
asLeakTesterTestEvaluation[83] := "TRANSDUCER VERIFY COMPLETE";
asLeakTesterTestEvaluation[84] := "ELEC REGULATOR CAL COMPLETE";
asLeakTesterTestEvaluation[85] := "ELEC REGULATOR CAL ERROR";
asLeakTesterTestEvaluation[86] := "SYSTEM ERROR - SERVICE REQ";
asLeakTesterTestEvaluation[87] := "TEST PORT SELECT CONFIG ERROR";
asLeakTesterTestEvaluation[88] := "SOURCE PRESSURE EXCEEDED";
asLeakTesterTestEvaluation[89] := "PRE-PRESSURE LOW";
asLeakTesterTestEvaluation[90] := "PRE-PRESSURE HIGH";
asLeakTesterTestEvaluation[91] := "ERROR: SNIFFER NOT READY";
asLeakTesterTestEvaluation[92] := "SNIFFER UNITS MISMATCH";
asLeakTesterTestEvaluation[93] := "SNIFFER MODE MISMATCH";
asLeakTesterTestEvaluation[94] := "T-GAS BACKGROUND FAULT";
asLeakTesterTestEvaluation[95] := "T-GAS MIN LEAK RATE FAULT";
asLeakTesterTestEvaluation[96] := "T-GAS CHAMBER CLEANUP FAULT";
asLeakTesterTestEvaluation[97] := "SNIFFER TYPE MISMATCH";
asLeakTesterTestEvaluation[98] := "SNIFFER READY INPUT FAULT";
asLeakTesterTestEvaluation[99] := "CHAMBER EVACUATION FAULT";
asLeakTesterTestEvaluation[100] := "CHAMBER RISE FAULT";
asLeakTesterTestEvaluation[101] := "SCALE CONFIG ERROR";
asLeakTesterTestEvaluation[102] := "SCALE NOT READY";
asLeakTesterTestEvaluation[103] := "SCALE NOT STABLE";
asLeakTesterTestEvaluation[104] := "SCALE WEIGHT LOW";
asLeakTesterTestEvaluation[105] := "SCALE WEIGHT HIGH";
asLeakTesterTestEvaluation[106] := "WEIGHT BELOW MIN";
asLeakTesterTestEvaluation[107] := "WEIGHT ABOVE MAX";
asLeakTesterTestEvaluation[108] := "ATMOSPHERIC PRESSURE COMPLETE";
asLeakTesterTestEvaluation[109] := "ATMOSPHERIC PRESSURE ERROR";
asLeakTesterTestEvaluation[110] := "EXTERNAL XDCR PRESS";
asLeakTesterTestEvaluation[111] := "MAN FILL SWITCH";
asLeakTesterTestEvaluation[112] := "ISOLATION FAILURE";
asLeakTesterTestEvaluation[113] := "LD ZERO < MIN";
asLeakTesterTestEvaluation[114] := "LD ZERO > MAX";
asLeakTesterTestEvaluation[115] := "LD LEAK < MIN";
asLeakTesterTestEvaluation[116] := "LD LEAK > MAX";
asLeakTesterTestEvaluation[117] := "PROCESS FAULT";
asLeakTesterTestEvaluation[118] := "POWER RESET";
asLeakTesterTestEvaluation[119] := "INVALID INPUT CONFIGURATION";
asLeakTesterTestEvaluation[120] := "INPUT INITIAL STATE ERROR";
asLeakTesterTestEvaluation[121] := "MASS SPEC CONTAMINATION";
asLeakTesterTestEvaluation[122] := "CHAMBER PRESSURE HIGH";
asLeakTesterTestEvaluation[123] := "CHAMBER CROSSOVER INPUT FAULT";
asLeakTesterTestEvaluation[124] := "CHAMBER RISE INPUT FAULT";
asLeakTesterTestEvaluation[125] := "T-GAS PART FILL FAULT";
asLeakTesterTestEvaluation[126] := "T-GAS LEAK STD FAULT";
asLeakTesterTestEvaluation[127] := "MASTER+LEAK LOSS<MIN M+L LOSS";
asLeakTesterTestEvaluation[128] := "LEAK LOSS<MIN LEAK LOSS";
asLeakTesterTestEvaluation[129] := "LEAK LOSS>MAX LEAK LOSS";
asLeakTesterTestEvaluation[130] := "MASTER+LEAK FLOW<MIN M+L FLOW";
asLeakTesterTestEvaluation[131] := "LEAK FLOW<MIN LEAK FLOW";
asLeakTesterTestEvaluation[132] := "LEAK FLOW > MAX LEAK FLOW";
asLeakTesterTestEvaluation[133] := "MASTER+LEAK PART COMPLETE";
asLeakTesterTestEvaluation[134] := "VALVE LOAD FAULT";
asLeakTesterTestEvaluation[135] := "ERROR: INSTRUMENT NOT ENABLED";
asLeakTesterTestEvaluation[136] := "CHARGE PRESSURE LOW";
asLeakTesterTestEvaluation[137] := "CHARGE PRESSURE HIGH";
END_ACTION

ACTION ACT_LeakTesterUnit:
asLeakTesterUnit[0] := "NO DATA";
asLeakTesterUnit[1] := "atm";
asLeakTesterUnit[2] := "bar";
asLeakTesterUnit[3] := "cmHg";
asLeakTesterUnit[4] := "inHg";
asLeakTesterUnit[5] := "kPa";
asLeakTesterUnit[6] := "MPa";
asLeakTesterUnit[7] := "mbar";
asLeakTesterUnit[8] := "mmHg";
asLeakTesterUnit[9] := "Pa";
asLeakTesterUnit[10] := "Torr";
asLeakTesterUnit[11] := "psig";
asLeakTesterUnit[12] := "psiv";
asLeakTesterUnit[13] := "iWC";
asLeakTesterUnit[14] := "cmWC";
asLeakTesterUnit[15] := "mmWC";
asLeakTesterUnit[16] := "ksc";
asLeakTesterUnit[17] := "psia";
asLeakTesterUnit[18] := "datm";
asLeakTesterUnit[19] := "dbar";
asLeakTesterUnit[20] := "dcmHg";
asLeakTesterUnit[21] := "dinHg";
asLeakTesterUnit[22] := "dkPa";
asLeakTesterUnit[23] := "dMpa";
asLeakTesterUnit[24] := "dmbar";
asLeakTesterUnit[25] := "dmmHg";
asLeakTesterUnit[26] := "dPa";
asLeakTesterUnit[27] := "dTorr";
asLeakTesterUnit[28] := "dpsig";
asLeakTesterUnit[29] := "dpsiv";
asLeakTesterUnit[30] := "diWC";
asLeakTesterUnit[31] := "dcmWC";
asLeakTesterUnit[32] := "dmmWC";
asLeakTesterUnit[33] := "dksc";
asLeakTesterUnit[34] := "dpsi";
asLeakTesterUnit[35] := "sccm";
asLeakTesterUnit[36] := "sces";
asLeakTesterUnit[37] := "scch";
asLeakTesterUnit[38] := "scfm";
asLeakTesterUnit[39] := "slpm";
asLeakTesterUnit[40] := "slps";
asLeakTesterUnit[41] := "scfh";
asLeakTesterUnit[42] := "scfs";
asLeakTesterUnit[43] := "slph";
asLeakTesterUnit[44] := "gs";
asLeakTesterUnit[45] := "gm";
asLeakTesterUnit[46] := "degC";
asLeakTesterUnit[47] := "degF";
asLeakTesterUnit[48] := "degK";
asLeakTesterUnit[49] := "hour";
asLeakTesterUnit[50] := "min";
asLeakTesterUnit[51] := "sec";
asLeakTesterUnit[52] := "msec";
asLeakTesterUnit[53] := "yr";
asLeakTesterUnit[54] := "mth";
asLeakTesterUnit[55] := "wk";
asLeakTesterUnit[56] := "day";
asLeakTesterUnit[57] := "cc";
asLeakTesterUnit[58] := "cin";
asLeakTesterUnit[59] := "l";
asLeakTesterUnit[60] := "gal";
asLeakTesterUnit[61] := "mL";
asLeakTesterUnit[62] := "in";
asLeakTesterUnit[63] := "mic";
asLeakTesterUnit[64] := "cm";
asLeakTesterUnit[65] := "mm";
asLeakTesterUnit[66] := "M";
asLeakTesterUnit[67] := "thou";
asLeakTesterUnit[68] := "mil";
asLeakTesterUnit[69] := "V";
asLeakTesterUnit[70] := "mV";
asLeakTesterUnit[71] := "uV";
asLeakTesterUnit[72] := "A";
asLeakTesterUnit[73] := "mA";
asLeakTesterUnit[74] := "uA";
asLeakTesterUnit[75] := "dB";
asLeakTesterUnit[76] := "bits";
asLeakTesterUnit[77] := "ppm";
asLeakTesterUnit[78] := "PF";
asLeakTesterUnit[79] := "%";
asLeakTesterUnit[80] := "unit";
asLeakTesterUnit[81] := "cnts";
asLeakTesterUnit[82] := "atm/s";
asLeakTesterUnit[83] := "bar/s";
asLeakTesterUnit[84] := "cHg/s";
asLeakTesterUnit[85] := "inHg/s";
asLeakTesterUnit[86] := "kPa/s";
asLeakTesterUnit[87] := "psi/s";
asLeakTesterUnit[88] := "iWC/s";
asLeakTesterUnit[89] := "cWC/s";
asLeakTesterUnit[90] := "mWC/s";
asLeakTesterUnit[91] := "ksc/s";
asLeakTesterUnit[92] := "g/a";
asLeakTesterUnit[93] := "oz/yr";
asLeakTesterUnit[94] := "ppm";
asLeakTesterUnit[95] := "mbl/s";
asLeakTesterUnit[96] := "Pam/s";
asLeakTesterUnit[97] := "acc/s";
asLeakTesterUnit[98] := "Trl/s";
asLeakTesterUnit[99] := "Pam/h";
asLeakTesterUnit[100] := "gr/yr";
asLeakTesterUnit[101] := "lb/yr";
asLeakTesterUnit[102] := "acc/m";
asLeakTesterUnit[103] := "kg";
asLeakTesterUnit[104] := "g";
asLeakTesterUnit[105] := "lb";
asLeakTesterUnit[106] := "oz";
asLeakTesterUnit[107] := "MPa/s";
asLeakTesterUnit[108] := "mb/s";
asLeakTesterUnit[109] := "mHg/s";
asLeakTesterUnit[110] := "pa/s";
asLeakTesterUnit[111] := "MPa/s";
END_ACTION

ACTION ACT_LiveSegmentCode:
asLeakTesterSegments[0] := "NO DATA";
asLeakTesterSegments[1] := "INTERN PreSeq";
asLeakTesterSegments[2] := "Intern PostSeq";
asLeakTesterSegments[3] := "Intern EmptySeq";
asLeakTesterSegments[4] := "Intern - Evaluate Part Result";
asLeakTesterSegments[5] := "Setup - Pre-Seq";
asLeakTesterSegments[6] := "Setup - Post-Seq";
asLeakTesterSegments[7] := "Setup - Pressure Select";
asLeakTesterSegments[8] := "Setup - Manifold Fill";
asLeakTesterSegments[9] := "Setup - Manifold Isolate";
asLeakTesterSegments[10] := "Setup - Manifold Exhaust";
asLeakTesterSegments[11] := "Prefill til Pressure";
asLeakTesterSegments[12] := "Prefill";
asLeakTesterSegments[13] := "Prefill Pre-Pressure";
asLeakTesterSegments[14] := "Prefill - Charge Volume";
asLeakTesterSegments[15] := "Fill References";
asLeakTesterSegments[16] := "Fill (without pressure monitoring)";
asLeakTesterSegments[17] := "Fill Ramp";
asLeakTesterSegments[18] := "Fill Tracer";
asLeakTesterSegments[19] := "Fill Tracer Gross";
asLeakTesterSegments[20] := "Fill Step";
asLeakTesterSegments[21] := "Fill Evac";
asLeakTesterSegments[22] := "Fill Clean";
asLeakTesterSegments[23] := "Fill til Full";
asLeakTesterSegments[24] := "Stabilize Tracer";
asLeakTesterSegments[25] := "Stabilize Tracer Gross";
asLeakTesterSegments[26] := "Stabilize DP Xder Balance";
asLeakTesterSegments[27] := "Stabilize Evac";
asLeakTesterSegments[28] := "Stabilize Step Dwell";
asLeakTesterSegments[29] := "Stabilize Chamber Cleanup";
asLeakTesterSegments[30] := "Stabilize til Slope";
asLeakTesterSegments[31] := "Stabilize DP";
asLeakTesterSegments[32] := "Stabilize Xder Test";
asLeakTesterSegments[33] := "Stabilize Flow";
asLeakTesterSegments[34] := "Stabilize References Volume";
asLeakTesterSegments[35] := "Stabilize Tracer Wait";
asLeakTesterSegments[36] := "Stabilize Balance DP";
asLeakTesterSegments[37] := "Pressure Decay - Leak Standard Test";
asLeakTesterSegments[38] := "Rate Pressure Loss Test";
asLeakTesterSegments[39] := "Occlusion Test (Backpressure)";
asLeakTesterSegments[40] := "Percent References Volume Test";
asLeakTesterSegments[41] := "Pressure Loss Test";
asLeakTesterSegments[42] := "Ramp Pressure Event Test";
asLeakTesterSegments[43] := "Proof Test";
asLeakTesterSegments[44] := "Ramp Flow Event Test";
asLeakTesterSegments[45] := "Refrigerant Fill";
asLeakTesterSegments[46] := "Ramp Digital Input Event Test";
asLeakTesterSegments[47] := "Sniffer Test";
asLeakTesterSegments[48] := "Sniffer Gross Test";
asLeakTesterSegments[49] := "Step Proof";
asLeakTesterSegments[50] := "Differential Pressure Decay - Leak Standard Test";
asLeakTesterSegments[51] := "Evac Test";
asLeakTesterSegments[52] := "Differential Pressure Decay Test";
asLeakTesterSegments[53] := "Differential Pressure Decay Test (no absl pressure)";
asLeakTesterSegments[54] := "Precise Mass Flow Test (Differential Flow)";
asLeakTesterSegments[55] := "Mass Flow Test";
asLeakTesterSegments[56] := "Mass Flow - Leak Rate Test";
asLeakTesterSegments[57] := "Differential Pressure Decay - Leak Standard Test (no absl pressure)";
asLeakTesterSegments[58] := "Differential Pressure Decay - Leak Rate (volume calculated)";
asLeakTesterSegments[59] := "Pressure Switch Test";
asLeakTesterSegments[60] := "Transducer Test";
asLeakTesterSegments[61] := "Pressure Verify";
asLeakTesterSegments[62] := "Exhaust";
asLeakTesterSegments[63] := "Exhaust til Pressure";
asLeakTesterSegments[64] := "Exhaust til Input";
asLeakTesterSegments[65] := "Exhaust til Analog Input";
asLeakTesterSegments[66] := "Exhaust til Slope";
asLeakTesterSegments[67] := "Exhaust til Empty";
asLeakTesterSegments[68] := "Exhaust - Re-Evacuate";
asLeakTesterSegments[69] := "Exhaust - T-Gas";
asLeakTesterSegments[70] := "Exhaust - Chamber Output Rest";
asLeakTesterSegments[71] := "Verify Pressure";
asLeakTesterSegments[72] := "Verify Pressure after Delay";
asLeakTesterSegments[73] := "Verify Input";
asLeakTesterSegments[74] := "Verify Input after Delay";
asLeakTesterSegments[75] := "Verify Analog Input";
asLeakTesterSegments[76] := "Verify Analog Input after Delay";
asLeakTesterSegments[77] := "Verify Slope";
asLeakTesterSegments[78] := "Verify Slope after Delay";
asLeakTesterSegments[79] := "Drive Output";
asLeakTesterSegments[80] := "Drive Output Period";
asLeakTesterSegments[81] := "Drive Analog Output";
asLeakTesterSegments[82] := "Drive Analog Output Period";
asLeakTesterSegments[83] := "Drive Valve";
asLeakTesterSegments[84] := "Drive Valve Period";
asLeakTesterSegments[85] := "Link Control";
asLeakTesterSegments[86] := "Link Decision";
asLeakTesterSegments[87] := "Autorun Relax";
asLeakTesterSegments[88] := "Calibration Relax";
asLeakTesterSegments[89] := "Delay";
asLeakTesterSegments[90] := "Pressure Transducer Zero";
asLeakTesterSegments[91] := "Flow Transducer Zero";
asLeakTesterSegments[92] := "Differential Pressure Transducer Zero";
asLeakTesterSegments[93] := "Pressure Select (Range Only)";
asLeakTesterSegments[94] := "Pressure Select (Evac)";
asLeakTesterSegments[95] := "Pressure Select";
asLeakTesterSegments[96] := "Pressure Select (Ramp)";
asLeakTesterSegments[97] := "Pressure Select (Tracer)";
asLeakTesterSegments[98] := "Pressure Select (Clean)";
asLeakTesterSegments[99] := "Pressure Select (None)";
asLeakTesterSegments[100] := "Tooling Motion Control";
asLeakTesterSegments[101] := "Tooling Motion Extend";
asLeakTesterSegments[102] := "Tooling Motion Retract";
asLeakTesterSegments[103] := "Tooling Part Mark";
asLeakTesterSegments[104] := "Tooling Seal Extend";
asLeakTesterSegments[105] := "Tooling Seal Retract";
asLeakTesterSegments[106] := "External Volume";
asLeakTesterSegments[107] := "Setup - Set Regulator";
asLeakTesterSegments[108] := "Setup - Electronic Regulator Analyze";
asLeakTesterSegments[109] := "Setup - Electronic Regulator Zero";
asLeakTesterSegments[110] := "Setup - Electronic Regulator Setpoint";
asLeakTesterSegments[111] := "Setup - Transducer Residual";
asLeakTesterSegments[112] := "Setup - Pressure Transducer Zero";
asLeakTesterSegments[113] := "Setup - Flow Transducer Zero";
asLeakTesterSegments[114] := "Setup - Pressure Transducer Setpoint";
asLeakTesterSegments[115] := "Setup - Flow Transducer Setpoint";
asLeakTesterSegments[116] := "Setup - DP Transducer Setpoint";
asLeakTesterSegments[117] := "Setup - Pressure Transducer Verification";
asLeakTesterSegments[118] := "Setup - Flow Transducer Verification";
asLeakTesterSegments[119] := "Setup - Sniffer Init 1";
asLeakTesterSegments[120] := "Setup - Sniffer Init 2";
asLeakTesterSegments[121] := "Setup - Sniffer Idle";
asLeakTesterSegments[122] := "Setup - Mix Verification";
asLeakTesterSegments[123] := "Setup - Scale Init";
asLeakTesterSegments[124] := "Setup - Atmospheric Pressure Check";
asLeakTesterSegments[125] := "Setup - DP Transducer Zero";
asLeakTesterSegments[126] := "Setup - DP Transducer Verification";
asLeakTesterSegments[127] := "Begin Chamber Functions";
asLeakTesterSegments[128] := "Chamber - hardvac control";
asLeakTesterSegments[129] := "Chamber - blower control";
asLeakTesterSegments[130] := "Chamber - inlet blower on";
asLeakTesterSegments[131] := "Chamber - inlet blower off";
asLeakTesterSegments[132] := "Chamber - circulation on";
asLeakTesterSegments[133] := "Chamber - outlet blower on";
asLeakTesterSegments[134] := "Chamber - outlet blower off";
asLeakTesterSegments[135] := "Chamber - circulation off";
asLeakTesterSegments[136] := "Chamber - accumulation rest";
asLeakTesterSegments[137] := "Chamber - clamshell purge rings control";
asLeakTesterSegments[138] := "Chamber - clamshell purge rings option";
asLeakTesterSegments[139] := "Chamber - clamshell purge rings rest";
asLeakTesterSegments[140] := "Chamber - Exh";
asLeakTesterSegments[141] := "Chamber - vent off";
asLeakTesterSegments[142] := "Chamber - evacuate on";
asLeakTesterSegments[143] := "Chamber - evacuate off";
asLeakTesterSegments[144] := "Chamber - pre-purge";
asLeakTesterSegments[145] := "Refrigerant CS Isolation";
asLeakTesterSegments[146] := "Refrigerant Stabilize";
asLeakTesterSegments[147] := "Refrigerant Part Switch";
asLeakTesterSegments[148] := "Refrigerant Vent";
asLeakTesterSegments[149] := "Refrigerant Iso Off";
asLeakTesterSegments[150] := "Stabilize Scale";
asLeakTesterSegments[151] := "Refrigerant Manual Fill";
asLeakTesterSegments[152] := "Refrigerant Evac";
END_ACTION

ACTION ACT_Precision:
asLeakTesterPrecision[0] := "NO DATA";
asLeakTesterPrecision[1] := "Digits of precision: X";
asLeakTesterPrecision[2] := "Digits of precision: X.X";
asLeakTesterPrecision[3] := "Digits of precision: X.XX";
asLeakTesterPrecision[4] := "Digits of precision: X.XXX";
asLeakTesterPrecision[5] := "Digits of precision: X.XXXX";
asLeakTesterPrecision[6] := "Digits of precision: X.XXXXX";
END_ACTION

ACTION ACT_ProgramEvaluation:
asLeakTesterProgramEvaluation[0] := "NO DATA";
asLeakTesterProgramEvaluation[1] := "TEST PASSED";
asLeakTesterProgramEvaluation[2] := "TEST FAILED";
asLeakTesterProgramEvaluation[3] := "TEST ERROR";
asLeakTesterProgramEvaluation[4] := "TEST SKIPPED";
asLeakTesterProgramEvaluation[5] := "TEST FAILED - LEVEL 1";
asLeakTesterProgramEvaluation[6] := "TEST FAILED - LEVEL 2";
asLeakTesterProgramEvaluation[7] := "TEST FAILED - LEVEL 3";
asLeakTesterProgramEvaluation[8] := "AUTO-CAL MASTER PART";
asLeakTesterProgramEvaluation[9] := "AUTO-CAL LEAK STANDARD PART";
asLeakTesterProgramEvaluation[10] := "TEST FAILED - NO EVENT";
asLeakTesterProgramEvaluation[11] := "TEST COMPLETE";
END_ACTION

ACTION ACT_TestType:
asLeakTesterTestType[0] := "NO DATA";
asLeakTesterTestType[1] := "Pressure Decay - Leak Standard Test";
asLeakTesterTestType[2] := "Rate of Pressure Loss Test";
asLeakTesterTestType[3] := "Occlusion Test (Backpressure)";
asLeakTesterTestType[4] := "Percent of Reference Volume Tes";
asLeakTesterTestType[5] := "Pressure Loss Test";
asLeakTesterTestType[6] := "Ramp to Pressure Event Test";
asLeakTesterTestType[7] := "Proof Test";
asLeakTesterTestType[8] := "Ramp to Flow Event Test";
asLeakTesterTestType[9] := "Refrigerant Fill";
asLeakTesterTestType[10] := "Ramp to Digital Input Event Test";
asLeakTesterTestType[11] := "Sniffer Test";
asLeakTesterTestType[12] := "";
asLeakTesterTestType[13] := "Sniffer Gross Test";
asLeakTesterTestType[14] := "Step Proof";
asLeakTesterTestType[15] := "Differential Pressure Decay - Leak | Standard Test";
asLeakTesterTestType[16] := "Evac Test";
asLeakTesterTestType[17] := "Differential Pressure Decay Test";
asLeakTesterTestType[18] := "Differential Pressure Decay Test (no abs pressure)";
asLeakTesterTestType[19] := "Precise Mass Flow Test (Differential Flow)";
asLeakTesterTestType[20] := "Mass Flow Test";
asLeakTesterTestType[21] := "Mass Flow - Leak Rate Test";
asLeakTesterTestType[22] := "Differential Pressure Decay - Leak Standard Test (no abs pressure)";
asLeakTesterTestType[23] := "Differential Pressure Decay - Leak Rate (volume calculated)";
asLeakTesterTestType[24] := "Pressure Switch Test";
asLeakTesterTestType[25] := "Transducer Test";
END_ACTION

END_PROGRAM

// ---- POUs/B_HightTest/PRG_HeightTest.TcPOU
PROGRAM PRG_HeightTest
VAR
	//FUNCTION
	fbHeightMeasurement2						: FB_HeightMeasurement2;
	
	
	
	bEnable										: BOOL;//
	bMeasurementRequest							: BOOL;//
	bAcknowledge								: BOOL;
	bBusy										: BOOL;//
	bComplete									: BOOL;//
	bEnableo									: BOOL;//
	bManualMode									: BOOL;
	
	bGreenIndicatorHeightTest	: BOOL;		     	
	bRedIndicatorHeightTest		: BOOL; 
	
//TrigTim

	rtrigCaseTriger			: ARRAY[1..20] OF R_TRIG;
	tonCaseDelay			: ARRAY[1..10] OF TON;
	
	
END_VAR


VAR_IN_OUT
	stStationStruct          	: ST_StandardStationStruct;
	
END_VAR
VAR PERSISTENT
stHeightMeasurement2						: ST_HeightMeasurement2;
stHeightlimit								: ST_Heightlimit;
END_VAR

ACT_IOLink();
ACT_TimTrig();
ACT_Statistics();
ACT_ProbesPosition();

(************** Station in Home Position **************************)
stStationStruct.bStationHomed :=  (stStationStruct.nState = 1000);

(******************************************************************)
stStationStruct.bStationComplete := stStationStruct.nState = 1220;
stStationStruct.bStationHomingRequest := stStationStruct.nState = 200;
stStationStruct.bStationWaitOnRequest := stStationStruct.nState = 1000; 
stStationStruct.bStationInitDone := stStationStruct.nState = 400;
stStationStruct.bStationInProgressInit := stStationStruct.nState >= 200 AND stStationStruct.nState <= 900;
stStationStruct.bStationInProgress :=  stStationStruct.nState > 1000 AND stStationStruct.nState < 1900;
stStationStruct.bStationWaitOnInit := stStationStruct.nState = 100; 
//stStationStruct.bStationAcknowledge := stStationStruct.nState = 200 OR stStationStruct.nState = 1100;
stStationStruct.bStationNotMoving := stStationStruct.nState = 100 OR stStationStruct.nState = 1000 OR stStationStruct.nState = 1240;
(******************************************************************)
(***************** Counter *************)


(***************************************)

IF rtrigCaseTriger[5].Q THEN
	stStationStruct.nState := 100;
END_IF

(***************************************)


CASE stStationStruct.nState OF
100:
bGreenIndicatorHeightTest	:= FALSE;		     	
bRedIndicatorHeightTest		:= FALSE; 
bMeasurementRequest := FALSE;
IF stStationStruct.bStationInitRequest THEN
	stStationStruct.nState:= 300;
END_IF

300:
IF tonCaseDelay[1].Q THEN
   stStationStruct.nState:= 400;	
END_IF
400:
	stStationStruct.nState:= 1000;

//============== Homed ========================================================

1000:

IF GVL_HMI_GLOBAL.bResetPassAndFail THEN
	bEnable 			:= FALSE;
	bAcknowledge 		:= FALSE;
	bMeasurementRequest	:= FALSE;
	GVL_MASTER.stNest.bHeightPass := FALSE;
	GVL_MASTER.stNest.sHeightHMI := "";
	GVL_MASTER.stNest.bHeightReject := FALSE;
	bGreenIndicatorHeightTest	:= FALSE;		 //    	
	bRedIndicatorHeightTest		:= FALSE; 		 //
END_IF
IF stStationStruct.bStationRequest AND stStationStruct.bNoCycleStopRequest THEN
   	stStationStruct.nState := 1010;  
ELSIF (stStationStruct.bStationManualRequestHMI OR GVL_MASTER.bManualModeTrigger) AND stStationStruct.bNoCycleStopRequest THEN
   stStationStruct.nState := 4000; // Manual Mode
ELSIF stStationStruct.bStationAbort THEN
	   stStationStruct.nState := 100;	   
END_IF
1010:
//bGreenIndicatorHeightTest	:= FALSE;		 //    	**LA 03/09/2025 Removed Because doesn't work the same tha leak station and added in line 60
//bRedIndicatorHeightTest		:= FALSE; 		 // 	**LA 03/09/2025 Removed Because doesn't work the same tha leak station and added in line 61
bEnable := TRUE;
IF tonCaseDelay[2].Q THEN
	stStationStruct.nState:= 1100;
END_IF
1100:
IF bEnableo THEN
	stStationStruct.nState:= 1110;
END_IF
1110:
bMeasurementRequest := TRUE;
IF NOT bBusy AND bComplete THEN
	bMeasurementRequest := FALSE;
	bAcknowledge		:= TRUE;
	stStationStruct.nState:= 1120;
END_IF
1120: // JOB PASS / JOB FAIL
bAcknowledge			:= FALSE;

IF tonCaseDelay[6].Q THEN
	
	GVL_MASTER.stNest.bHeightPass := GVL_HMI_GLOBAL.aGeneralPassHeightTest[5];
	GVL_MASTER.stNest.bHeightReject := GVL_HMI_GLOBAL.aGeneralFailHeightTest[5];
	
	IF GVL_MASTER.stNest.bHeightPass THEN
		GVL_MASTER.stNest.sHeightHMI 	:= "Pass";
		GVL_MASTER.stNest.bHeightPass := TRUE;
		GVL_MASTER.stNest.bHeightReject := FALSE;
		bGreenIndicatorHeightTest	:= TRUE;		     	
		bRedIndicatorHeightTest		:= FALSE; 
	ELSIF  GVL_MASTER.stNest.bHeightReject THEN
		
		GVL_MASTER.stNest.sHeightHMI 	:= "Fail";
		GVL_MASTER.stNest.bHeightPass := FALSE;
		GVL_MASTER.stNest.bHeightReject := TRUE;
		bGreenIndicatorHeightTest	:= FALSE;		     	
		bRedIndicatorHeightTest		:= TRUE; 
	END_IF
	
	stStationStruct.nState:= 1220;
END_IF
1220:

IF tonCaseDelay[5].Q THEN
	stStationStruct.nState:= 1240;
END_IF

1240:
IF (tonCaseDelay[3].Q AND  GVL_MASTER.bHeightTestacknowledge) OR NOT stStationStruct.bNoCycleStopRequest THEN	
	stStationStruct.nState:= 1000;
END_IF
4000://Manual Mode

IF NOT stStationStruct.bStationManualRequestHMI  THEN
   stStationStruct.nState := 1000;
   bManualMode					:= FALSE;
	bEnable						:= FALSE; 
ELSIF stStationStruct.bStationAbort THEN
	   stStationStruct.nState := 100;
	   bManualMode					:= FALSE;
		bEnable						:= FALSE;
ELSE 
	bManualMode					:= TRUE;
	bEnable						:= TRUE;  
END_IF
END_CASE

ACTION ACT_IOLink:

stHeightMeasurement2.aSensorCurrentValue[1]		:= DINT_TO_REAL(GVL_IO.dw_B08_DL_PN1.gt2_1_1CurrentValue);
stHeightMeasurement2.aSensorCurrentValue[2]		:= DINT_TO_REAL(GVL_IO.dw_B08_DL_PN1.gt2_1_2CurrentValue);
stHeightMeasurement2.aSensorCurrentValue[3]		:= DINT_TO_REAL(GVL_IO.dw_B08_DL_PN1.gt2_1_3CurrentValue);
stHeightMeasurement2.aSensorCurrentValue[4]		:= DINT_TO_REAL(GVL_IO.dw_B08_DL_PN1.gt2_2CurrentValue);

fbHeightMeasurement2(
	
	aSensorCurrentValue							:= stHeightMeasurement2.aSensorCurrentValue,	
	bEnable										:= bEnable,
	bMeasurementRequest							:= bMeasurementRequest,
	bSetFixedPoints								:= GVL_HMI_GLOBAL.bSetSetPointsHeightTest,
	aTolerance									:= stHeightMeasurement2.aTolerance,
	bAcknowledge								:= bAcknowledge,
	nDistanceBetweenPoints						:= stHeightMeasurement2.nDistanceBetweenPoints,
	anDistanceSetPoint							:= stHeightMeasurement2.anDistanceSetPoint,
	bManualMode									:= bManualMode,
	
	//OUTPUTS
	bBusy										=> bBusy,
	bComplete									=> bComplete,
	bEnableo									=> bEnableo,
	aPass										=> GVL_HMI_GLOBAL.aGeneralPassHeightTest ,
	aFail										=> GVL_HMI_GLOBAL.aGeneralFailHeightTest ,
	aMinLimitCalibrationBlock					=> stHeightMeasurement2.aMinLimitCalibrationBlock,
	aMaxLimitCalibrationBlock					=> stHeightMeasurement2.aMaxLimitCalibrationBlock,
	aDistanceBetweenProbes						=> stHeightMeasurement2.aDistanceBetweenProbes,
	abSensorStuck								=> stHeightMeasurement2.abSensorStuck,
	nFixedPoint									=> stHeightMeasurement2.nFixedPoint,
	aScaledSensorCurrentValue					=> stHeightMeasurement2.aScaledSensorCurrentValue,
	nHeightMeasureStateValue					=> GVL_HMI_GLOBAL.nHeightMeasureStateValue);


IF NOT stStationStruct.bNoCycleStopRequest OR stStationStruct.bStationAbort THEN
	GVL_MASTER.bHeightTestacknowledge := TRUE;
END_IF

GVL_HMI_GLOBAL.nHeightTestCycTime := (TIME_TO_DINT(GVL_MASTER.stAlarms[1].aEventTimers[11].ET))/1000;

//to save data 
GVL_MASTER.stNest.nDistance							:= stHeightMeasurement2.aDistanceBetweenProbes;
GVL_MASTER.stNest.nTarget							:= stHeightMeasurement2.anDistanceSetPoint;
END_ACTION

ACTION ACT_ProbesPosition:
IF ((stHeightMeasurement2.aScaledSensorCurrentValue[1]> stHeightlimit.LOW)  AND 
	(stHeightMeasurement2.aScaledSensorCurrentValue[1]<stHeightlimit.HIGH)) AND	
   ((stHeightMeasurement2.aScaledSensorCurrentValue[2]>stHeightlimit.LOW)  AND 
	(stHeightMeasurement2.aScaledSensorCurrentValue[2]<stHeightlimit.HIGH)) AND
   ((stHeightMeasurement2.aScaledSensorCurrentValue[3]>stHeightlimit.LOW)  AND 
	(stHeightMeasurement2.aScaledSensorCurrentValue[3]<stHeightlimit.HIGH)) AND
   ((stHeightMeasurement2.aScaledSensorCurrentValue[4]>stHeightlimit.LOW)  AND 
	(stHeightMeasurement2.aScaledSensorCurrentValue[4]<stHeightlimit.HIGH)) THEN

		GVL_HMI_GLOBAL.bProbesPositionOk				:= TRUE;
ELSE 	GVL_HMI_GLOBAL.bProbesPositionOk				:= FALSE;		
	
END_IF
END_ACTION

ACTION ACT_Statistics:

//GENERAL
IF rtrigCaseTriger[3].Q THEN
GVL_PERSIST.stPartsInspection.nHeightPartsGood:= GVL_PERSIST.stPartsInspection.nHeightPartsGood +1;
GVL_PERSIST.stPartsInspection.nHeightTotalPartsGood := GVL_PERSIST.stPartsInspection.nHeightTotalPartsGood+1;
ELSIF GVL_HMI_GLOBAL.bResetHeightGoodParts THEN
GVL_PERSIST.stPartsInspection.nHeightPartsGood:=0;	
END_IF


IF rtrigCaseTriger[4].Q THEN
	GVL_PERSIST.stPartsInspection.nHeightPartsFailed:=GVL_PERSIST.stPartsInspection.nHeightPartsFailed + 1;
	GVL_PERSIST.stPartsInspection.nHeightTotalPartsFailed:= GVL_PERSIST.stPartsInspection.nHeightTotalPartsFailed + 1;
ELSIF GVL_HMI_GLOBAL.bResetHeightFailParts THEN
	GVL_PERSIST.stPartsInspection.nHeightPartsFailed:=0;
END_IF


//Distance 1

IF rtrigCaseTriger[6].Q THEN
GVL_PERSIST.stPartsInspection.nHeightDistancePartsGood[1]:= GVL_PERSIST.stPartsInspection.nHeightDistancePartsGood[1] +1;
GVL_PERSIST.stPartsInspection.nHeightDistanceTotalPartsGood[1] := GVL_PERSIST.stPartsInspection.nHeightDistanceTotalPartsGood[1]+1;
ELSIF GVL_HMI_GLOBAL.aResetHeightSensorGoodParts[1] THEN
GVL_PERSIST.stPartsInspection.nHeightDistancePartsGood[1]:=0;	
END_IF


IF rtrigCaseTriger[7].Q THEN
	GVL_PERSIST.stPartsInspection.nHeightDistancePartsFailed[1]:=GVL_PERSIST.stPartsInspection.nHeightDistancePartsFailed[1] + 1;
	GVL_PERSIST.stPartsInspection.nHeightDistanceTotalPartsFailed[1]:= GVL_PERSIST.stPartsInspection.nHeightDistanceTotalPartsFailed[1] + 1;
ELSIF GVL_HMI_GLOBAL.aResetHeightSensorBadParts[1] THEN
	GVL_PERSIST.stPartsInspection.nHeightDistancePartsFailed[1]:=0;
END_IF

//Distance 2

IF rtrigCaseTriger[8].Q THEN
GVL_PERSIST.stPartsInspection.nHeightDistancePartsGood[2]:= GVL_PERSIST.stPartsInspection.nHeightDistancePartsGood[2] +1;
GVL_PERSIST.stPartsInspection.nHeightDistanceTotalPartsGood[2] := GVL_PERSIST.stPartsInspection.nHeightDistanceTotalPartsGood[2]+1;
ELSIF GVL_HMI_GLOBAL.aResetHeightSensorGoodParts[2] THEN
GVL_PERSIST.stPartsInspection.nHeightDistancePartsGood[2]:=0;	
END_IF


IF rtrigCaseTriger[9].Q THEN
	GVL_PERSIST.stPartsInspection.nHeightDistancePartsFailed[2]:=GVL_PERSIST.stPartsInspection.nHeightDistancePartsFailed[2] + 1;
	GVL_PERSIST.stPartsInspection.nHeightDistanceTotalPartsFailed[2]:= GVL_PERSIST.stPartsInspection.nHeightDistanceTotalPartsFailed[2] + 1;
ELSIF GVL_HMI_GLOBAL.aResetHeightSensorBadParts[2] THEN
	GVL_PERSIST.stPartsInspection.nHeightDistancePartsFailed[2]:=0;
END_IF

//Distance 3

IF rtrigCaseTriger[10].Q THEN
GVL_PERSIST.stPartsInspection.nHeightDistancePartsGood[3]:= GVL_PERSIST.stPartsInspection.nHeightDistancePartsGood[3] +1;
GVL_PERSIST.stPartsInspection.nHeightDistanceTotalPartsGood[3] := GVL_PERSIST.stPartsInspection.nHeightDistanceTotalPartsGood[3]+1;
ELSIF GVL_HMI_GLOBAL.aResetHeightSensorGoodParts[3] THEN
GVL_PERSIST.stPartsInspection.nHeightDistancePartsGood[3]:=0;	
END_IF


IF rtrigCaseTriger[11].Q THEN
	GVL_PERSIST.stPartsInspection.nHeightDistancePartsFailed[3]:=GVL_PERSIST.stPartsInspection.nHeightDistancePartsFailed[3] + 1;
	GVL_PERSIST.stPartsInspection.nHeightDistanceTotalPartsFailed[3]:= GVL_PERSIST.stPartsInspection.nHeightDistanceTotalPartsFailed[3] + 1;
ELSIF GVL_HMI_GLOBAL.aResetHeightSensorBadParts[3] THEN
	GVL_PERSIST.stPartsInspection.nHeightDistancePartsFailed[3]:=0;
END_IF
END_ACTION

ACTION ACT_TimTrig:
tonCaseDelay[1](IN:= (stStationStruct.nState=300),PT:=T#50MS);
tonCaseDelay[2](IN:= (stStationStruct.nState=1010),PT:=T#800MS);
tonCaseDelay[3](IN:= (stStationStruct.nState=1240),PT:=T#100MS);
tonCaseDelay[4](IN:=bMeasurementRequest ,PT:=T#1S);
tonCaseDelay[5](IN:=stStationStruct.nState=1220 ,PT:=T#2S);
tonCaseDelay[6](IN:= stStationStruct.nState=1120 AND GVL_HMI_GLOBAL.aGeneralPassHeightTest[5] <> GVL_HMI_GLOBAL.aGeneralFailHeightTest[5] ,PT:=T#250MS);
tonCaseDelay[7](IN:= ,PT:=T#50MS);
tonCaseDelay[8](IN:= ,PT:=T#250MS);
tonCaseDelay[9](IN:= ,PT:=T#250MS);
tonCaseDelay[10](IN:= ,PT:=T#250MS);

rtrigCaseTriger[1](clk:= );
rtrigCaseTriger[2](clk:= );
rtrigCaseTriger[3](clk:= (stStationStruct.nState=1240) AND GVL_MASTER.stNest.bHeightPass );//
rtrigCaseTriger[4](clk:= (stStationStruct.nState=1240) AND GVL_MASTER.stNest.bHeightReject );//
rtrigCaseTriger[5](clk:= stStationStruct.bStationAbort);
rtrigCaseTriger[6](clk:= (stStationStruct.nState=1240) AND GVL_HMI_GLOBAL.aGeneralPassHeightTest[1]);
rtrigCaseTriger[7](clk:= (stStationStruct.nState=1240) AND GVL_HMI_GLOBAL.aGeneralFailHeightTest[1]);
rtrigCaseTriger[8](clk:= (stStationStruct.nState=1240) AND GVL_HMI_GLOBAL.aGeneralPassHeightTest[2]);
rtrigCaseTriger[9](clk:= (stStationStruct.nState=1240) AND GVL_HMI_GLOBAL.aGeneralFailHeightTest[2]);
rtrigCaseTriger[10](clk:= (stStationStruct.nState=1240) AND GVL_HMI_GLOBAL.aGeneralPassHeightTest[3]);
rtrigCaseTriger[11](clk:= (stStationStruct.nState=1240) AND GVL_HMI_GLOBAL.aGeneralFailHeightTest[3]);
rtrigCaseTriger[12](clk:=);
rtrigCaseTriger[13](clk:= );
END_ACTION

END_PROGRAM

// ---- POUs/G_Utility/FB_HeightMeasurement2.TcPOU
FUNCTION_BLOCK FB_HeightMeasurement2
VAR_INPUT
	
	aSensorCurrentValue							: ARRAY[1..4] OF REAL;		
	bEnable										: BOOL;
	bMeasurementRequest							: BOOL;
	bManualMode									: BOOL;
	bSetFixedPoints								: BOOL;
	aTolerance									: ARRAY[1..3] OF REAL;
	
	bAcknowledge								: BOOL;
	
	//Calibration block
	
	nDistanceBetweenPoints						: ARRAY[1..3] OF REAL;
	anDistanceSetPoint							: ARRAY[1..3] OF REAL;
	
	
	
	
					
END_VAR
VAR_OUTPUT
	
	bBusy										: BOOL;
	bComplete									: BOOL;
	bEnableo									: BOOL;
	aPass										: ARRAY[1..5] OF BOOL; //5 Final Result
	aFail										: ARRAY[1..5] OF BOOL; //5 Final Result
	aMinLimitCalibrationBlock					: ARRAY[1..3] OF REAL;
	aMaxLimitCalibrationBlock					: ARRAY[1..3] OF REAL;
	
	aDistanceBetweenProbes						: ARRAY[1..3] OF REAL; //1 Probe 1 to probe zero
	abSensorStuck								: ARRAY[1..4] OF BOOL;
	nFixedPoint									: ARRAY[1..4] OF REAL;
	aScaledSensorCurrentValue					: ARRAY[1..4] OF REAL;
	
	nHeightMeasureStateValue					: ARRAY[1..4] OF DINT;

	

END_VAR
VAR PERSISTENT
	
	nSensorSetPoint								: ARRAY[1..4] OF REAL;
	
END_VAR
VAR
	
	i											: INT;
	j											: INT;
	tonTestingTime								: TON;
	rMeasurementRequest							: R_TRIG;
	nHeightOffset								: REAL;
	
	EHeighttMeasureProcess						: E_HeighttMeasureProcess;
	anValueBeforeMeasurement					: ARRAY[1..4] OF REAL;
	
	
END_VAR

ACT_ScaleMinMax();
ACT_SetPoints();

IF NOT bEnable THEN
	EHeighttMeasureProcess						:= E_HeighttMeasureProcess.WAITING_ENABLE;
ELSIF bManualMode AND bEnable THEN
	EHeighttMeasureProcess						:= E_HeighttMeasureProcess.Manual_Mode;
END_IF
bEnableo										:= bEnable;
tonTestingTime( IN := (EHeighttMeasureProcess = E_HeighttMeasureProcess.WAITING_FOR_MEASURE), PT := T#3S);
rMeasurementRequest( CLK := bMeasurementRequest);

CASE EHeighttMeasureProcess OF

E_HeighttMeasureProcess.WAITING_ENABLE:

	IF bEnable THEN
		EHeighttMeasureProcess					:= E_HeighttMeasureProcess.WAITING_MEASURING_REQUEST;
	END_IF

E_HeighttMeasureProcess.WAITING_MEASURING_REQUEST:	

	bComplete									:= FALSE;
	IF rMeasurementRequest.Q THEN
		EHeighttMeasureProcess					:= E_HeighttMeasureProcess.RESET;
	END_IF
	
	anValueBeforeMeasurement					:= aSensorCurrentValue;

E_HeighttMeasureProcess.RESET:
	
	
	abSensorStuck[1]							:= FALSE;
	
	FOR i := 1 TO 5 DO
		aPass[i]								:= FALSE;	
		aFail[i]								:= FALSE;
	END_FOR
	FOR j := 1 TO 3 DO
		nHeightMeasureStateValue[j]				:= 0;
	END_FOR
		EHeighttMeasureProcess					:= E_HeighttMeasureProcess.WAITING_FOR_MEASURE;
	
E_HeighttMeasureProcess.SENSOR_STUCK_EVALUATION:

	ACT_SensorStuck();
	
E_HeighttMeasureProcess.WAITING_FOR_MEASURE:

	IF tonTestingTime.Q  THEN
		EHeighttMeasureProcess					:= E_HeighttMeasureProcess.CALIBRATIONBLOCK_METHOD;
	END_IF

E_HeighttMeasureProcess.CALIBRATIONBLOCK_METHOD:

		ACT_CalibrationBlockMethod();
		bComplete								:= TRUE;
		IF bAcknowledge THEN
			EHeighttMeasureProcess					:= E_HeighttMeasureProcess.WAITING_MEASURING_REQUEST;
		END_IF

E_HeighttMeasureProcess.Manual_Mode:
		
		ACT_ManualMode();		

END_CASE


bBusy				:= 	(EHeighttMeasureProcess	<> E_HeighttMeasureProcess.WAITING_ENABLE AND
						EHeighttMeasureProcess  <> E_HeighttMeasureProcess.WAITING_MEASURING_REQUEST) AND
						NOT bComplete;

ACTION ACT_CalibrationBlockMethod:
aDistanceBetweenProbes[1] 	:= (nFixedPoint[4] - aScaledSensorCurrentValue[4])+ (aScaledSensorCurrentValue[1] - (nFixedPoint[1])) + nDistanceBetweenPoints[1];
aDistanceBetweenProbes[2] 	:= (nFixedPoint[4] - aScaledSensorCurrentValue[4])+ (aScaledSensorCurrentValue[2] - (nFixedPoint[2])) + nDistanceBetweenPoints[2];
aDistanceBetweenProbes[3] 	:= (nFixedPoint[4] - aScaledSensorCurrentValue[4])+ (aScaledSensorCurrentValue[3] - (nFixedPoint[3])) + nDistanceBetweenPoints[3];

FOR i := 1 TO 3 DO
	IF (aDistanceBetweenProbes[i] <= aMaxLimitCalibrationBlock[i]) AND (aDistanceBetweenProbes[i] >= aMinLimitCalibrationBlock[i]) THEN
		
		aPass[i]			:= TRUE;
		nHeightMeasureStateValue[i] := 1;
	ELSE 
		aFail[i]			:= TRUE;
		nHeightMeasureStateValue[i] := 2;
	END_IF
END_FOR

IF aPass[1] AND aPass[2] AND aPass[3] THEN
	aPass[5]			:= TRUE;
ELSIF aFail[1] OR aFail[2] OR aFail[3] THEN
	aFail[5]			:= TRUE;
END_IF
END_ACTION

ACTION ACT_ManualMode:
aDistanceBetweenProbes[1] 	:= (nFixedPoint[4] - aScaledSensorCurrentValue[4])+ (aScaledSensorCurrentValue[1] - (nFixedPoint[1])) + nDistanceBetweenPoints[1];
aDistanceBetweenProbes[2] 	:= (nFixedPoint[4] - aScaledSensorCurrentValue[4])+ (aScaledSensorCurrentValue[2] - (nFixedPoint[2])) + nDistanceBetweenPoints[2];
aDistanceBetweenProbes[3] 	:= (nFixedPoint[4] - aScaledSensorCurrentValue[4])+ (aScaledSensorCurrentValue[3] - (nFixedPoint[3])) + nDistanceBetweenPoints[3];

IF (aDistanceBetweenProbes[1] <= aMaxLimitCalibrationBlock[1]) AND (aDistanceBetweenProbes[1] >= aMinLimitCalibrationBlock[1]) THEN
	
		nHeightMeasureStateValue[1] := 1;
ELSE 
		nHeightMeasureStateValue[1] := 2;
END_IF

IF (aDistanceBetweenProbes[2] <= aMaxLimitCalibrationBlock[2]) AND (aDistanceBetweenProbes[2] >= aMinLimitCalibrationBlock[2]) THEN
	
		nHeightMeasureStateValue[2] := 1;
ELSE 
		nHeightMeasureStateValue[2] := 2;
END_IF

IF (aDistanceBetweenProbes[3] <= aMaxLimitCalibrationBlock[3]) AND (aDistanceBetweenProbes[3] >= aMinLimitCalibrationBlock[3]) THEN
	
		nHeightMeasureStateValue[3] := 1;
ELSE 
		nHeightMeasureStateValue[3] := 2;
END_IF
END_ACTION

ACTION ACT_ScaleMinMax:
//Current value SCALE
IF aSensorCurrentValue[1] <> 0 THEN
	
	aScaledSensorCurrentValue[1]		:= aSensorCurrentValue[1]/10000;
	
ELSE aScaledSensorCurrentValue[1]		:= 0;

END_IF

IF aSensorCurrentValue[2] <> 0 THEN
	
	aScaledSensorCurrentValue[2]		:= aSensorCurrentValue[2]/10000;
	
ELSE aScaledSensorCurrentValue[2]		:= 0;

END_IF

IF aSensorCurrentValue[3] <> 0 THEN
	
	aScaledSensorCurrentValue[3]		:= aSensorCurrentValue[3]/10000;
	
ELSE aScaledSensorCurrentValue[3]		:= 0;

END_IF

IF aSensorCurrentValue[4] <> 0 THEN
	
	aScaledSensorCurrentValue[4]		:= aSensorCurrentValue[4]/10000;
	
ELSE aScaledSensorCurrentValue[4]		:= 0;

END_IF

aMaxLimitCalibrationBlock[1]			:= anDistanceSetPoint[1] + aTolerance[1];
aMaxLimitCalibrationBlock[2]			:= anDistanceSetPoint[2] + aTolerance[2];
aMaxLimitCalibrationBlock[3]			:= anDistanceSetPoint[3] + aTolerance[3];

aMinLimitCalibrationBlock[1]			:= anDistanceSetPoint[1] - aTolerance[1];
aMinLimitCalibrationBlock[2]			:= anDistanceSetPoint[2] - aTolerance[2];
aMinLimitCalibrationBlock[3]			:= anDistanceSetPoint[3] - aTolerance[3];
END_ACTION

ACTION ACT_SensorStuck:
IF (anValueBeforeMeasurement[1] <= (aSensorCurrentValue[1] + 0.5)) AND (anValueBeforeMeasurement[1] >= (aSensorCurrentValue[1] - 0.5)) THEN
		abSensorStuck[1]							:= TRUE;
	END_IF

IF (anValueBeforeMeasurement[2] <= (aSensorCurrentValue[2] + 0.5)) AND (anValueBeforeMeasurement[2] >= (aSensorCurrentValue[2] - 0.5)) THEN
		abSensorStuck[2]							:= TRUE;
	END_IF

IF (anValueBeforeMeasurement[3] <= (aSensorCurrentValue[3] + 0.5)) AND (anValueBeforeMeasurement[3] >= (aSensorCurrentValue[3] - 0.5)) THEN
		abSensorStuck[3]							:= TRUE;
	END_IF

IF (anValueBeforeMeasurement[4] <= (aSensorCurrentValue[4] + 0.5)) AND (anValueBeforeMeasurement[4] >= (aSensorCurrentValue[4] - 0.5)) THEN
		abSensorStuck[4]							:= TRUE;
	END_IF
END_ACTION

ACTION ACT_SetPoints:
IF bSetFixedPoints THEN
	
	nSensorSetPoint[1]						:= aScaledSensorCurrentValue[1];
	nSensorSetPoint[2]						:= aScaledSensorCurrentValue[2];
	nSensorSetPoint[3]						:= aScaledSensorCurrentValue[3];
	nSensorSetPoint[4]						:= aScaledSensorCurrentValue[4];
	
	
ELSE
	
	nFixedPoint[1]							:= nSensorSetPoint[1];
	nFixedPoint[2]							:= nSensorSetPoint[2];
	nFixedPoint[3]							:= nSensorSetPoint[3];
	nFixedPoint[4]							:= nSensorSetPoint[4];

END_IF
END_ACTION

END_FUNCTION_BLOCK
